IF xEmergenciaOK THEN
	//se nao tiver bloqueado
	IF NOT xBloqueado THEN
		//tudo que da pra considerar uma falha
		IF (NOT xFalha) THEN
			IF xLigaManu OR (xLigaManu3S AND NOT Ton3Segundos.q) THEN
				xCmdFWD := TRUE;
			ELSE
				xCmdFWD := FALSE;
			END_IF
		END_IF
	END_IF
END_IF

IF (xReset OR xResetBlocoComunicacao) AND xFalha THEN
	xCmdFWD := xCmdRev := FALSE;
END_IF

// joga a velo normal nele 
iVelocidade := real_to_int(rSetPoinManu);

//protege contra numeros negativos ou divisao por 0
IF stMotor.Config.xVeloEmPorcentagem THEN
	rSetPoinManu := 100;

	IF stMotor.Config.rVeloEmPorcentagem_VeloMax < 0.1 THEN
		stMotor.Config.rVeloEmPorcentagem_VeloMax := 1;
	END_IF

	iVelocidade := TO_INT((rSetPoinManu * stMotor.Config.rVeloEmPorcentagem_VeloMax) / 100);
END_IF

IF stMotor.Config.xVeloEmMetroPMin THEN
	//rSetPoinManu := 1800;
	//protege contra numeros negativos ou divisao por 0
	IF stMotor.Config.rVeloEmMetroPMin_Conversao < 0.1 THEN
		stMotor.Config.rVeloEmMetroPMin_Conversao := 1;
	END_IF

	iVelocidade := 1800;//TO_INT((rSetPoinManu * 1800) / stMotor.Config.rVeloEmMetroPMin_Conversao);
END_IF

// se tiver que inverte a velo e tiver comissionado
IF stMotor.Config.xInverteSentido THEN
	//se o operador meter uma velo negativva nao da BO
	IF iVelocidade < 0 THEN
		iVelocidade := iVelocidade;
	ELSE
		iVelocidade := iVelocidade * -1;
	END_IF

END_IF

xLigado := (xCmdFwd OR xCmdRev) AND xFazendoComissionamento;
END_ACTION

ACTION Falhas:

xResetParaInversor := xReset OR xResetBlocoComunicacao;

IF xReset OR xResetBlocoComunicacao THEN
	xFalhaContatora := FALSE;
	xFalhaPartidaSoft := FALSE;
END_IF

rtVoltouOnline(CLK := xInversorOnline, Q =>);

IF rtVoltouOnline.q THEN
	xFalha	:= FALSE;
	xReset	:= TRUE;
END_IF

TON_Partida(IN := ((xCmdFwd OR xCmdRev) AND NOT ((xContatorLigado OR xByPassContator)) AND xTemContatora),
			PT := REAL_TO_TIME(stMotor.Config.rTempoFeedBackContator * 1000),
			Q =>,
			ET =>);

IF TON_Partida.q THEN
	xFalhaContatora := TRUE;
END_IF

// as condiçoes que geram falha
xFalha := FALSE;

// se nao vier o sinal da contatora
IF xFalhaContatora THEN
	xFalha := TRUE OR xFalha;
END_IF

//Disjuntor desarmado
IF (NOT xDisjuntorOK AND NOT xByPassDisjuntor) AND xTemDisjuntor THEN
	xFalha := TRUE OR xFalha;
END_IF

// se o inversor nao ficar online
IF ((xTemInversor OR xTemTeSysU) AND (NOT xInversorOnline AND NOT xBypassRede)) THEN
	xFalha := TRUE OR xFalha;
END_IF

//se o inversor entrar em falha
IF ((xTemInversor OR xTemTeSysU) AND (xFalhaInversor AND NOT xBypassRede)) THEN
	xFalha := TRUE OR xFalha;
END_IF

//se o inversor entrar em falha
IF (xTemContatoInversorOK AND ((NOT xContatoInversorOK) AND NOT xBypassContatoInversorOK)) THEN
	xFalha := TRUE OR xFalha;
END_IF

//se o freio nao vier
IF (NOT xFreioOK AND NOT xBypassFreio) AND stMotor.Config.xTemFreio THEN
	xFalha := TRUE OR xFalha;
END_IF


TON_soft
	(
		IN := (xCmdFwd OR xCmdRev) AND NOT (xContatoRodandoSoft OR xBypassContatorunSoft) AND stMotor.Config.xTemSoft,
			PT := REAL_TO_TIME(stMotor.Config.rTempoDeRampaSoft * 1000),
			Q =>,
			ET =>);

IF TON_soft.q THEN
	xFalhaPartidaSoft := TRUE;
END_IF

IF xFalhaPartidaSoft THEN
	xFalha := TRUE OR xFalha;
END_IF

IF xSoftEmFalhaCOM AND NOT xBypassSoftEmFalhaCOM THEN
	xFalha := TRUE OR xFalha;
END_IF

//se o inversor entrar em falha
IF ((xContatoFalhaSoft) AND NOT stMotor.Config.xBypassContatoFalhaSoft) AND stMotor.Config.xTemSoft THEN
	xFalha := TRUE OR xFalha;
END_IF

//se foi detectada uma falta de fase
IF NOT xFaltaDeFaseOk THEN
	xFalha := TRUE OR xFalha;
END_IF
END_ACTION

METHOD FB_init : BOOL
VAR_INPUT
	bInitRetains	: BOOL;	// if TRUE, the retain variables are initialized (warm start / cold start)
	bInCopyCode		: BOOL;	// if TRUE, the instance afterwards gets moved into the copy code (online change)
END_VAR

(*
IF bInCopyCode THEN
	
	IF CHK_REAL(stMotor.Config.iSetPoinManu) <> 0 THEN
		stMotor.Config.iSetPoinManu := 0;
	END_IF
	
	IF CHK_REAL(stMotor.Config.rCorrente_Comissionada) <> 0 THEN
		stMotor.Config.rCorrente_Comissionada := 0;
	END_IF
	
	IF CHK_REAL(stMotor.Config.rSetPoinAuto) <> 0 THEN
		stMotor.Config.rSetPoinAuto := 0;
	END_IF
	
	IF CHK_REAL(stMotor.Config.rTempoFeedBackContator) <> 0 THEN
		stMotor.Config.rTempoFeedBackContator := 0;
	END_IF
	
	IF CHK_REAL(stMotor.Config.rTempoProxMotor) <> 0 THEN
		stMotor.Config.rTempoProxMotor := 0;
	END_IF
	
	IF CHK_REAL(stMotor.Config.rTempoTrocaSentidoDeMarcha) <> 0 THEN
		stMotor.Config.rTempoTrocaSentidoDeMarcha := 0;
	END_IF
	
	IF CHK_REAL(stMotor.Config.rVeloEmMetroPMin_Conversao) <> 0 THEN
		stMotor.Config.rVeloEmMetroPMin_Conversao := 0;
	END_IF
	
	IF (stMotor.Config.xByPassContator) <> TRUE AND (stMotor.Config.xByPassContator) <> FALSE THEN
		stMotor.Config.xByPassContator := FALSE;
	END_IF
	
	IF (stMotor.Config.xByPassDisjuntor) <> TRUE AND (stMotor.Config.xByPassDisjuntor) <> FALSE THEN
		stMotor.Config.xByPassDisjuntor := FALSE;
	END_IF
	
	IF (stMotor.Config.xBypassRede) <> TRUE AND (stMotor.Config.xBypassRede) <> FALSE THEN
		stMotor.Config.xBypassRede := FALSE;
	END_IF
	
	IF (stMotor.Config.xComissionado_Corrente) <> TRUE AND (stMotor.Config.xComissionado_Corrente) <> FALSE THEN
		stMotor.Config.xComissionado_Corrente := FALSE;
	END_IF
	
	IF (stMotor.Config.xComissionado_Sentido) <> TRUE AND (stMotor.Config.xComissionado_Sentido) <> FALSE THEN
		stMotor.Config.xComissionado_Sentido := FALSE;
	END_IF
	
	IF (stMotor.Config.xComissionado_Velo) <> TRUE AND (stMotor.Config.xComissionado_Velo) <> FALSE THEN
		stMotor.Config.xComissionado_Velo := FALSE;
	END_IF
	
	IF (stMotor.Config.xInverteSentido) <> TRUE AND (stMotor.Config.xInverteSentido) <> FALSE THEN
		stMotor.Config.xInverteSentido := FALSE;
	END_IF
	
	IF (stMotor.Config.xTemReversao) <> TRUE AND (stMotor.Config.xTemReversao) <> FALSE THEN
		stMotor.Config.xTemReversao := FALSE;
	END_IF
	
	IF (stMotor.Config.xVeloEmMetroPMin) <> TRUE AND (stMotor.Config.xVeloEmMetroPMin) <> FALSE THEN
		stMotor.Config.xVeloEmMetroPMin := FALSE;
	END_IF
	
	IF (stMotor.Config.xVeloEmPorcentagem) <> TRUE AND (stMotor.Config.xVeloEmPorcentagem) <> FALSE THEN
		stMotor.Config.xVeloEmPorcentagem := FALSE;
	END_IF

END_IF
*)
END_METHOD

ACTION FirstScan:




//Ultima_stMotor		:= stMotor;
rSetPoinManu		:= stMotor.Config.rSetPoinManu;
rSetPoinAuto		:= stMotor.Config.rSetPoinAuto;
xByPassContator		:= stMotor.Config.xByPassContator;
xByPassDisjuntor	:= stMotor.Config.xByPassDisjuntor;

FOR i := 0 TO 23 DO
	stMotor.KPI[i].stGraficoIHM[0].x := 'Desligado';
	stMotor.KPI[i].stGraficoIHM[0].sCor := '#555555';
	stMotor.KPI[i].stGraficoIHM[0].y := 100;
	
	stMotor.KPI[i].stGraficoIHM[1].x := 'Ligado';
	stMotor.KPI[i].stGraficoIHM[1].sCor := '#F1F1F1';
	
	stMotor.KPI[i].stGraficoIHM[2].x := 'Interlok';
	stMotor.KPI[i].stGraficoIHM[2].sCor := '#FFFF00';
	
	stMotor.KPI[i].stGraficoIHM[3].x := 'Falha';
	stMotor.KPI[i].stGraficoIHM[3].sCor := '#FF0000';
	
	stMotor.KPI[i].stGraficoIHM[4].x := 'Emergencia';
	stMotor.KPI[i].stGraficoIHM[4].sCor := '#CC0000';
END_FOR
END_ACTION

ACTION Horimetro:
(*// aqui ta o lendario codigo que no incendo do frigorifico de rolandia diminuiu de 30 para 15 o uso da CPU, chupa mundo
// muito inificiente //Total chad de codigo
systime(timeLoDw => currentTime.dwLowDateTime, timeHiDW => currentTime.dwHighDateTime);

dtAux := FILETIME_TO_DT(currentTime)-(T#3H);
timeStructAux := DT_TO_SYSTEMTIME(dtAux);
*)

fbHorimetro(xConta := stMotor.Sa.xCmdFwd OR stMotor.Sa.xCmdRev,
			xReset := stHoraAgora.wDay <> wDiaAnterior,
			Tempo => tHorimetro,
			stHoraAgora := stHoraAgora);

wDiaAnterior := stHoraAgora.wDay;

sHorimetro := F_TempoEmStringAteHoras
	(
		Tempo := tHorimetro,
			xMostraHoras := TRUE,
			xMostraMinutos := TRUE,
			xMostraSegundos := TRUE,
			xMostraMilisegundos := FALSE,
			xCascata := FALSE);

stMotor.Sa.sHorimetro	:= sHorimetro;
stMotor.Sa.tHorimetro	:= tHorimetro;
END_ACTION

ACTION KPI:

rtLigou(CLK:=xLigado);
IF rtLigou.q THEN
	IF xLigado THEN
		stMotor.KPI[0].iVezesLigado := stMotor.KPI[0].iVezesLigado + 1;
	ELSE
		stMotor.KPI[0].iVezesdesligado := stMotor.KPI[0].iVezesdesligado + 1;
	END_IF
END_IF

rtfalha(CLK:=xFalha);
IF rtfalha.q THEN
	stMotor.KPI[0].iVezesFalha := stMotor.KPI[0].iVezesFalha + 1;
END_IF

rtEmergencia(CLK:=xEmergenciaOK);
IF rtEmergencia.q THEN
	stMotor.KPI[0].iVezesEmergencia := stMotor.KPI[0].iVezesEmergencia + 1;
END_IF

rtInterlock(CLK:=xParadoPorInterlock);
IF rtInterlock.q THEN
	stMotor.KPI[0].iVezesInterlock := stMotor.KPI[0].iVezesInterlock + 1;
END_IF



IF wSegAnterior <> stHoraAgora.wSecond THEN

	IF xFalha AND xEmergenciaOK THEN
		stMotor.KPI[0].rPorcFalha	:= stMotor.KPI[0].rPorcFalha + 0.027777;
		stMotor.KPI[0].tFalha		:= stMotor.KPI[0].tFalha + T#1S;
	END_IF

	IF NOT xEmergenciaOK THEN
		stMotor.KPI[0].rPorcEmergencia	:= stMotor.KPI[0].rPorcEmergencia + 0.027777;
		stMotor.KPI[0].tEmergencia		:= stMotor.KPI[0].tEmergencia + T#1S;
	END_IF

	IF xParadoPorInterlock THEN
		stMotor.KPI[0].rPorcInterlock	:= stMotor.KPI[0].rPorcInterlock + 0.027777;
		stMotor.KPI[0].tInterlock		:= stMotor.KPI[0].tInterlock + T#1S;
	END_IF

	IF xCmdFwd THEN
		stMotor.KPI[0].rPorcLigado	:= stMotor.KPI[0].rPorcLigado + 0.027777;
		stMotor.KPI[0].tLigado		:= stMotor.KPI[0].tLigado + T#1S;
	END_IF
	
	
	// Pro OEE Fechar ele precisa considerar so o tempo que ele deveria estar ligado
	IF xLigaAuto THEN // Para o OEE
		tTempoComxLigaAuto		:= tTempoComxLigaAuto + T#1S;
	END_IF
	
	IF xLigaAuto AND NOT xEmergenciaOK THEN // Para o OEE
		tXligaEEmergencia		:= tXligaEEmergencia + T#1S;
	END_IF
	
	IF xLigaAuto AND xParadoPorInterlock THEN // Para o OEE
		tXligaEInterlock		:= tXligaEInterlock + T#1S;
	END_IF
	
	IF xLigaAuto AND xFalha AND xEmergenciaOK THEN // Para o OEE
		tXligaEFalha			:= tXligaEFalha + T#1S;
	END_IF
	
	

	stMotor.KPI[0].rPorcDesligado :=
		100 - stMotor.KPI[0].rPorcLigado - stMotor.KPI[0].rPorcInterlock - stMotor.KPI[0].rPorcEmergencia - stMotor.KPI[0].rPorcFalha;

	stMotor.KPI[0].tDesligado :=
		T#1H - stMotor.KPI[0].tLigado - stMotor.KPI[0].tInterlock - stMotor.KPI[0].tEmergencia - stMotor.KPI[0].tFalha;
		
	rAux := DINT_TO_REAL(TRUNC(stMotor.KPI[0].rPorcDesligado*100));
	stMotor.KPI[0].stGraficoIHM[0].y := rAux/100;
	rAux := DINT_TO_REAL(TRUNC(stMotor.KPI[0].rPorcLigado*100));
	stMotor.KPI[0].stGraficoIHM[1].y := rAux/100;
	rAux := DINT_TO_REAL(TRUNC(stMotor.KPI[0].rPorcInterlock*100));
	stMotor.KPI[0].stGraficoIHM[2].y := rAux/100;
	rAux := DINT_TO_REAL(TRUNC(stMotor.KPI[0].rPorcFalha*100));
	stMotor.KPI[0].stGraficoIHM[3].y := rAux/100;
	rAux := DINT_TO_REAL(TRUNC(stMotor.KPI[0].rPorcEmergencia*100));
	stMotor.KPI[0].stGraficoIHM[4].y := rAux/100;
	


END_IF

IF whoraAnterior <> stHoraAgora.wHour THEN
	
	//OEE
	udiLigado 		:= TIME_TO_UDINT(tTempoComxLigaAuto);
	udiFalha 		:= TIME_TO_UDINT(tXligaEFalha);
	udiEmergencia 	:= TIME_TO_UDINT(tXligaEEmergencia);
	udiinterlock 	:= TIME_TO_UDINT(tXligaEInterlock);
	
	
	rAux1 := (udiLigado-udiFalha);
	IF udiLigado <> 0 THEN
		rAux1 := rAux1/udiLigado; // disponibilidade em valor
		stMotor.KPI[0].rDisponibilidade := rAux1 * 100;
	ELSE
		stMotor.KPI[0].rDisponibilidade := 0;
	END_IF
	
	rAux1 := (udiLigado-udiFalha-udiEmergencia-udiinterlock);
	rAux2 := (udiLigado-udiFalha);
	IF rAux2 <> 0 THEN
		rAux1 := rAux1/rAux2; // Performace em valor
		stMotor.KPI[0].rPerformace := rAux1 * 100;
	ELSE
		stMotor.KPI[0].rPerformace := 0;
	END_IF
	
	
	stMotor.KPI[0].rQualidade := 100;
	stMotor.KPI[0].rOEE := (stMotor.KPI[0].rDisponibilidade * stMotor.KPI[0].rPerformace * stMotor.KPI[0].rQualidade) / 10000;
	
	
	
	stMotor.KPI[0].stGraficoDisponibilidade[0].x := 'Disponivel';
	stMotor.KPI[0].stGraficoDisponibilidade[0].sCor := '#32CD32';
	stMotor.KPI[0].stGraficoDisponibilidade[0].label := ' ';
	stMotor.KPI[0].stGraficoDisponibilidade[0].y := stMotor.KPI[0].rDisponibilidade;
	
	stMotor.KPI[0].stGraficoDisponibilidade[0].x := 'Indisponivel';
	stMotor.KPI[0].stGraficoDisponibilidade[0].sCor := '#FFFFFF00';
	stMotor.KPI[0].stGraficoDisponibilidade[0].label := ' ';
	stMotor.KPI[0].stGraficoDisponibilidade[0].y := 100 - stMotor.KPI[0].rDisponibilidade;
	
	
	stMotor.KPI[0].stGraficoPerformace[0].x := 'Performando';
	stMotor.KPI[0].stGraficoPerformace[0].sCor := '#32CD32';
	stMotor.KPI[0].stGraficoPerformace[0].label := ' ';
	stMotor.KPI[0].stGraficoPerformace[0].y := stMotor.KPI[0].rPerformace;
	
	stMotor.KPI[0].stGraficoPerformace[0].x := 'Não performando';
	stMotor.KPI[0].stGraficoPerformace[0].sCor := '#FFFFFF00';
	stMotor.KPI[0].stGraficoPerformace[0].label := ' ';
	stMotor.KPI[0].stGraficoPerformace[0].y := 100 - stMotor.KPI[0].rPerformace;
	
	
	stMotor.KPI[0].stGraficoQualidade[0].x := 'Qualidade';
	stMotor.KPI[0].stGraficoQualidade[0].sCor := '#32CD32';
	stMotor.KPI[0].stGraficoQualidade[0].label := ' ';
	stMotor.KPI[0].stGraficoQualidade[0].y := stMotor.KPI[0].rQualidade;
	
	stMotor.KPI[0].stGraficoQualidade[0].x := 'Mal qualidade';
	stMotor.KPI[0].stGraficoQualidade[0].sCor := '#FFFFFF00';
	stMotor.KPI[0].stGraficoQualidade[0].label := ' ';
	stMotor.KPI[0].stGraficoQualidade[0].y := 100 - stMotor.KPI[0].rQualidade;
	
	
	stMotor.KPI[0].stGraficoOEE[0].x := 'OEE';
	stMotor.KPI[0].stGraficoOEE[0].sCor := '#32CD32';
	stMotor.KPI[0].stGraficoOEE[0].label := ' ';
	stMotor.KPI[0].stGraficoOEE[0].y := stMotor.KPI[0].rOEE;
	
	stMotor.KPI[0].stGraficoOEE[0].x := 'OEE ruim';
	stMotor.KPI[0].stGraficoOEE[0].sCor := '#FFFFFF00';
	stMotor.KPI[0].stGraficoOEE[0].label := ' ';
	stMotor.KPI[0].stGraficoOEE[0].y := 100 - stMotor.KPI[0].rOEE;
	
	
	
	
	//KPI NORMAL


	FOR i := 23 TO 1 BY -1 DO
		stMotor.KPI[i] := stMotor.KPI[i - 1];
	END_FOR

	stMotor.KPI[0] := kpiVazio;
	tTempoComxLigaAuto := T#0S;
	tXligaEEmergencia := T#0S;
	tXligaEFalha := T#0S;
	tXligaEInterlock := T#0S;
	
	stMotor.KPI[0].stGraficoIHM[0].x := 'Desligado';
	stMotor.KPI[0].stGraficoIHM[0].sCor := '#555555';
	stMotor.KPI[0].stGraficoIHM[0].label := ' ';
	stMotor.KPI[0].stGraficoIHM[0].y := 100;
	
	stMotor.KPI[0].stGraficoIHM[1].x := 'Ligado';
	stMotor.KPI[0].stGraficoIHM[1].label := ' ';
	stMotor.KPI[0].stGraficoIHM[1].sCor := '#F1F1F1';
	
	stMotor.KPI[0].stGraficoIHM[2].x := 'Interlok';
	stMotor.KPI[0].stGraficoIHM[2].label := ' ';
	stMotor.KPI[0].stGraficoIHM[2].sCor := '#FFFF00';
	
	stMotor.KPI[0].stGraficoIHM[3].x := 'Falha';
	stMotor.KPI[0].stGraficoIHM[3].label := ' ';
	stMotor.KPI[0].stGraficoIHM[3].sCor := '#FF0000';
	
	stMotor.KPI[0].stGraficoIHM[4].x := 'Emergencia';
	stMotor.KPI[0].stGraficoIHM[4].label := ' ';
	stMotor.KPI[0].stGraficoIHM[4].sCor := '#CC0000';
END_IF

whoraAnterior	:= stHoraAgora.wHour;
wSegAnterior	:= stHoraAgora.wSecond;
END_ACTION

ACTION ProxMotor:

/// Liga prox motor na sequencia

// se tiver o comando pra ligar ele ja manda essa e se tiver inversor ele ajeita ali em baixo
tonLigaProxMotor.IN := (xCmdFwd OR xCmdRev) AND NOT xFalha;

//se tiver inversor
IF xTemInversor AND (xCmdFwd OR xCmdRev) THEN
	//se o inversor mandar que velo ele ta
	IF stMotor.LeiturasInversorIHM.sVelocidadeRPM <> ''
			AND stMotor.LeiturasInversorIHM.sVelocidadeRPM <> 'NA'
			AND stMotor.LeiturasInversorIHM.sVelocidadeRPM <> 'ND' THEN
		tonLigaProxMotor.IN :=xCmdFwd; // AND NOT xFalha;		
	END_IF
END_IF

tonLigaProxMotor(PT := REAL_TO_TIME(stMotor.Config.rTempoProxMotor * 1000), Q => , ET =>);

xNaoLigaProxMotor := NOT tonLigaProxMotor.q;
END_ACTION

ACTION SegurancaReversao:

//Prende eles em falso para o motor esperar trocar o sentido de giro

xTrocandoSentido := FALSE;
//lembrando que tp funciona na base do pulso , entao faz sentido ser assim
tpTrocaSentidoDeRotacao(IN :=, PT := REAL_TO_TIME(stMotor.Config.rTempoTrocaSentidoDeMarcha * 1000), Q =>, ET =>);

IF tpTrocaSentidoDeRotacao.q AND xLigado THEN
	xCmdFWD := xCmdRev	:= FALSE;
	xTrocandoSentido	:= TRUE;
END_IF

//Controle caso ele troque o sentido 
tpTrocaSentidoDeRotacao.IN := FALSE;

btTrocouSentidoRotAuto(CLK := xReversoAuto AND stMotor.Config.xTemReversao, Q =>);

IF btTrocouSentidoRotAuto.q THEN
	IF xCmdFwd OR xCmdRev THEN
		IF xAutomaticoManual THEN
			tpTrocaSentidoDeRotacao.IN := TRUE;
		END_IF
	END_IF
END_IF

btTrocouSentidoRotManu(CLK := xReversoManu AND stMotor.Config.xTemReversao, Q =>);

IF btTrocouSentidoRotManu.q THEN
	IF xCmdFwd OR xCmdRev THEN
		IF NOT xAutomaticoManual THEN
			tpTrocaSentidoDeRotacao.IN := TRUE;
		END_IF
	END_IF
END_IF

btTrocouManualAutomatico(CLK := xAutomaticoManual AND stMotor.Config.xTemReversao, Q =>);

IF btTrocouManualAutomatico.q THEN
	IF xReversoAuto <> xReversoManu THEN
		tpTrocaSentidoDeRotacao.IN := TRUE;
	END_IF
END_IF
END_ACTION

ACTION Status:

//STAUTS
IF (NOT xCmdFwd OR NOT xCmdrev) AND NOT xBloqueado AND xEmergenciaOK THEN
	IF xAutomaticoManual THEN
		iStsMotor := 1; // parado em automatico
		sStatus := 'Parado em automatico';
	ELSE
		iStsMotor := 2; // parado em manual
		sStatus := 'Parado em manual';
	END_IF
END_IF

IF (xCmdFwd OR xCmdrev) AND (NOT xBloqueado OR xEmergenciaOK) THEN
	IF xAutomaticoManual THEN
		iStsMotor := 3; // rodando em automatico
		sStatus := 'Rodando em automatico';
	ELSE
		iStsMotor := 4; // rodando em manual
		sStatus := 'Rodando em manual';
	END_IF
END_IF

IF stMotor.En.xLigaHigienizacao AND xHabilitaHigienizacao THEN
	iStsMotor := 18; // Higienização Ligada
	sStatus := 'Rodando Higienização';
END_IF

IF stMotor.En.xLigaHigienizacao AND NOT xHabilitaHigienizacao THEN
	iStsMotor := 17; // Higienização Parado
	sStatus := 'Parado Higienização';
END_IF

IF xParadoPorInterlock THEN
	iStsMotor := 10; // Parado por interlock
	sStatus := 'Parado por interlock';
END_IF

IF xTrocandoSentido THEN
	iStsMotor := 11; // Trocando sentido
	sStatus := 'trocando sentido de giro';
END_IF

IF xBloqueado THEN
	iStsMotor := 5; // bloquado
	sStatus := 'Bloqueado';
END_IF

IF xFalhaContatora THEN
	iStsMotor := 6; // em falha na partida
	sStatus := 'Falha contatora';
END_IF

IF ((xTemInversor OR xTemTeSysU) AND (NOT xInversorOnline AND NOT xBypassRede)) THEN
	iStsMotor := 7; // em inversor offline
	IF xTemInversor THEN
		sStatus := 'Inversor offline';
	ELSE
		sStatus := 'TeSysU offline';
	END_IF
END_IF

IF ((xTemInversor OR xTemTeSysU) AND (xFalhaInversor AND NOT xBypassRede)) THEN
	iStsMotor := 12; // Inversor em falha
	IF xTemInversor THEN
		sStatus := 'Falha COM. inversor';
	ELSE
		sStatus := 'Falha COM. TeSysU';
	END_IF
END_IF

IF (xTemContatoInversorOK AND (NOT (xContatoInversorOK) AND NOT xBypassContatoInversorOK)) THEN
	iStsMotor := 14; // Inversor Sem o contato de OK
	sStatus := 'Falha contato inversor';
END_IF

IF NOT xDisjuntorOK AND NOT xByPassDisjuntor AND xTemDisjuntor THEN
	iStsMotor := 8; // disjuntor desarmado
	sStatus := 'Disjuntor desarmado';
END_IF

IF (stMotor.Config.xTemFreio AND (NOT xFreioOK AND NOT xBypassFreio)) THEN
	iStsMotor := 13; // disjuntor desarmado
	sStatus := 'Disjuntor desarmado';
END_IF

IF xFalhaPartidaSoft THEN
	iStsMotor := 15; // em falha na partida da soft
	sStatus := 'Falha na partida da soft';
END_IF

IF ((xContatoFalhaSoft)) AND stMotor.Config.xTemSoft THEN
	iStsMotor := 16; // em falha na soft
	sStatus := 'Falha contato soft';
END_IF

IF ((xSoftEmFalhaCOM)) AND stMotor.Config.xBypassSoftEmFalhaCOM THEN
	iStsMotor := 19; // em falha na soft
	sStatus := 'Falha COM. soft';
END_IF


IF NOT xFaltaDeFaseOk THEN
	iStsMotor := 20; // Falta de fase detectada
	sStatus := 'falta de fase';
END_IF

IF NOT xEmergenciaOK THEN
	iStsMotor := 9; // emergencia
	sStatus := 'Emergencia';
END_IF
END_ACTION

END_FUNCTION_BLOCK

// POUs/Siemens/SinaSpeed/Sina_SpeedV2
FUNCTION_BLOCK Sina_SpeedV2
VAR_IN_OUT
	motor : st_Partida;
END_VAR
VAR_INPUT
	EnableAxis	:	BOOL;//	0	Non-RETAIN	TRUE	TRUE	TRUE	FALSE	0-->1; 1 = Enable the drive (OFF2 / OFF 3 are 1 in default status) (OFF1 = 0-->1)
	AckError	:	BOOL;//	0	Non-RETAIN	TRUE	TRUE	TRUE	FALSE	1 = Acknowledge drive error
	SpeedSp		:	REAL;//	0.0	Non-retain	True	True	True	False	Speed standardises with the standardisation factor
	RefSpeed	:	REAL;//	0.0	Non-retain	True	True	True	False	Standardisation factor of speed
	ConfigAxis	:	Word_Bits;//	Non-RETAIN	TRUE	TRUE	TRUE	FALSE	binary programmed input TO control all functions in the telegram without its own FUNCTION block input
	HWIDZSW AT %I* 	:	InversorSinaSpeed;//	Non-retain	True	True	True	False	Hardware Identifer set point slot
END_VAR
VAR_OUTPUT
	AxisEnabled	:	BOOL;//	0	Non-RETAIN	TRUE	TRUE	TRUE	FALSE	1 = Drive is enabled
	Lockout		:	BOOL;//	0	Non-RETAIN	TRUE	TRUE	TRUE	FALSE	1 = Drive lockout active
	ActVelocity	:	REAL;//	0.0	Non-RETAIN	TRUE	TRUE	TRUE	FALSE	Actual in [U/MIN]
	Error		:	BOOL;//	0	Non-RETAIN	TRUE	TRUE	TRUE	FALSE	1 = Error  (FB AND Infeed)
	Status		:	WORD;//	0	Non-RETAIN	TRUE	TRUE	TRUE	FALSE	Status output (7002 = FB in operation; 8xxx = error description  - read the manual)
	DiagId		:	WORD;//	16#0000	Non-RETAIN	TRUE	TRUE	TRUE	FALSE	Error codes OF the cyclic system funtion blocks DPWR / DPRD_DAT
	HWIDSTW AT %Q*	:	Inversor_2Words_SinaSpeed;//	Non-retain	True	True	True	False	Hardware Identifer actual value slot
	Corrente 	: REAL;
	Potencia 	: REAL;
	Torque 		: REAL;
	ErroAtual 	: UINT;
END_VAR
VAR
	sxSendBuf	:	sxSendBuf;//		Non-RETAIN	TRUE	TRUE	TRUE	FALSE	Send buffer
	sxRecvBuf	:	sxRecvBuf;//		Non-RETAIN	TRUE	TRUE	TRUE	FALSE	Receive buffer

	piRetSFC	:	INT;//						Status FOR fault analysis
	piCount		:	INT;//							Freely available counter variable 3
	prVelocity	:	REAL;//							velocity
	pdRecvBuf	:	DWORD;//							Buffer OF Recv-Value
	pdSendBuf	:	DWORD;//							Buffer OF Send-Value
	phLAddr		:	InversorSinaSpeed;//							Start addr FROM the I/O process image area OF MOD (DEC) FOR DPWR_DAT/DPRD_DAT
	swSendBuf	:	ARRAY[0..1] OF WORD;//							Sendepuffer
	swRecvBuf	:	ARRAY[0..1] OF WORD;//							Empfangspuffer         Static variables
	
	//Adicionado por Tiago
	xPrimeiroScan : BOOL := TRUE;
END_VAR


//=============================================================================
//SIEMENS AG
//(c)Copyright 2017 All Rights Reserved
//-----------------------------------------------------------------------------
// Library: DriveLib
// Tested with: S7-1516-3 PN/DP V1.8
// Engineering: TIA Portal V14
// Restrictions: -
// Requirements: S7-1200 / S7-1500
// Functionality: cyclic communication between a SINAMICS a PLC.
//                If in HWConfig Std.TLG 1 is projected 2 PZD-words are exchanged
//                in every bus cycle.
//                The parametrisation of these words is described in the manual of the
//                SINAMICS
//=============================================================================

//Adicionado por Tiago
IF xPrimeiroScan THEN
	ConfigAxis.wor := 63;
	xPrimeiroScan := FALSE;
END_IF


EnableAxis := motor.Sa.xCmdFwd;
AckError := motor.Sa.xResetParaInversor;
SpeedSp := motor.Sa.iVelocidade;





Corrente := HWIDZSW.StatusWord2.ui16b * 25.0 / 16384; // 2.5 = parametro interno
Torque := HWIDZSW.StatusWord3.ui16b * 58.36 / 16384; // parametro interno
Potencia := HWIDZSW.StatusWord4.ui16b * 11.0 / 16384; // parametro interno
ErroAtual := HWIDZSW.StatusWord5.ui16b;

motor.LeiturasInversorIHM.sVelocidadeRPM := concat(TO_STRING(F_RetiraCasa(Entrada:= ActVelocity, casa:= 1)),' RPM');
motor.LeiturasInversorIHM.sCorrente := concat(TO_STRING(F_RetiraCasa(Entrada:= Corrente, casa:= 2)),' A');
motor.LeiturasInversorIHM.sTorque := concat(TO_STRING(F_RetiraCasa(Entrada:= Torque, casa:= 2)),' Nm');
motor.LeiturasInversorIHM.sVelocidadeHz := concat(TO_STRING(F_RetiraCasa(Entrada:= Potencia, casa:= 2)),' KW');
motor.LeiturasInversorIHM.sUltimoErro := TO_STRING(DiagId);

// Fim adicionado por tiago

















// Schreibdaten zusammenstellen
// Steuerword aufbereiten

sxSendBuf.STW1.x16b.bBit0 := EnableAxis;
sxSendBuf.STW1.x16b.bBit1 := ConfigAxis.bits.bBit0;
sxSendBuf.STW1.x16b.bBit2 := ConfigAxis.bits.bBit1;
sxSendBuf.STW1.x16b.bBit3 := ConfigAxis.bits.bBit2;
sxSendBuf.STW1.x16b.bBit4 := ConfigAxis.bits.bBit3;
sxSendBuf.STW1.x16b.bBit5 := ConfigAxis.bits.bBit4;
sxSendBuf.STW1.x16b.bBit6 := ConfigAxis.bits.bBit5;
sxSendBuf.STW1.x16b.bBit10 := TRUE;
sxSendBuf.STW1.x16b.bBit11 := ConfigAxis.bits.bBit6;
sxSendBuf.STW1.x16b.bBit7 := AckError;

// Geschwindigkeit
IF RefSpeed <> 0 THEN
  prVelocity := SpeedSp * (16384.0 / RefSpeed);
  // Limit REAL - Variable to INT - Limits
  IF prVelocity > 32767 THEN
    prVelocity := 32767;
  ELSIF prVelocity < -32768 THEN
    prVelocity := -32768;
  ELSE
    ; // not needed
  END_IF;
  sxSendBuf.Velocity.Valor := INT_TO_WORD(REAL_TO_INT(prVelocity));
  
ELSE
  sxSendBuf.Velocity.Valor := 16#0;
END_IF;
swSendBuf[0] := sxSendBuf.STW1.ui16b;
swSendBuf[1] := UDINT_TO_WORD(sxSendBuf.Velocity.Valor);

//Prozessdaten zur Signalbaugruppe schreiben
(*
piRetSFC := DPWR_DAT(LADDR := HWIDSTW,
                      RECORD := swSendBuf);
*)

piRetSFC := 0;

HWIDSTW.StatusWord0.ui16b := swSendBuf[0];
HWIDSTW.StatusWord1.ui16b := swSendBuf[1];





// Fehler der RÃ¼ckmeldung ausgeben
DiagId := INT_TO_WORD(piRetSFC);

//kein Fehler beim Schreiben
IF piRetSFC = 0 THEN
  
  //kein Fehler beim Schreiben
  IF piRetSFC = 0 THEN
    
    //Prozessdaten von der Signalbaugruppe lesen
	(*
    #piRetSFC := DPRD_DAT(LADDR := #HWIDZSW,
                          RECORD => #swRecvBuf);
						  *)
	
	piRetSFC := 0;
						  
	swRecvBuf[0] := HWIDZSW.StatusWord0.ui16b;
	swRecvBuf[1] := HWIDZSW.StatusWord1.ui16b;			
    
    // Fehler der RÃ¼ckmeldung ausgeben
    DiagId := INT_TO_WORD(piRetSFC);
  END_IF;
  
  //Fehler beim Lesen (Profibus-Kommunikation unterbrochen)
  IF piRetSFC <> 0 THEN
    
    // Fehler
    Error := TRUE;
    Status := 16#8600;
    
    // Zustandsworte lÃ¶schen
    sxRecvBuf.ZSW1.x16b.bBit8 := 0;
    sxRecvBuf.ZSW1.x16b.bBit9 := 0;
    sxRecvBuf.ZSW1.x16b.bBit10 := 0;
    sxRecvBuf.ZSW1.x16b.bBit11 := 0;
    sxRecvBuf.ZSW1.x16b.bBit12 := 0;
    sxRecvBuf.ZSW1.x16b.bBit13 := 0;
    sxRecvBuf.ZSW1.x16b.bBit14 := 0;
    sxRecvBuf.ZSW1.x16b.bBit15 := 0;
    sxRecvBuf.ZSW1.x16b.bBit0 := 0;
    sxRecvBuf.ZSW1.x16b.bBit1 := 0;
    sxRecvBuf.ZSW1.x16b.bBit2 := 0;
    sxRecvBuf.ZSW1.x16b.bBit3 := 0;
    sxRecvBuf.ZSW1.x16b.bBit4 := 0;
    sxRecvBuf.ZSW1.x16b.bBit5 := 0;
    sxRecvBuf.ZSW1.x16b.bBit6 := 0;
    sxRecvBuf.ZSW1.x16b.bBit7 := 0;
    
    
    (*#sxRecvBuf.sxZSW1.SpDev   := 0;
    #sxRecvBuf.sxZSW1.Pcd     := 0;
    #sxRecvBuf.sxZSW1.Comp    := 0;
    #sxRecvBuf.sxZSW1.CurLim  := 0;
    #sxRecvBuf.sxZSW1.Brake   := 0;
    #sxRecvBuf.sxZSW1.Motover := 0;
    #sxRecvBuf.sxZSW1.Dir     := 0;
    #sxRecvBuf.sxZSW1.Invover := 0;
    #sxRecvBuf.sxZSW1.Rts     := 0;
    #sxRecvBuf.sxZSW1.Rdy     := 0;
    #sxRecvBuf.sxZSW1.IOp     := 0;
    #sxRecvBuf.sxZSW1.Fault   := 0;
    #sxRecvBuf.sxZSW1.NoOff2  := 0;
    #sxRecvBuf.sxZSW1.NoOff3  := 0;
    #sxRecvBuf.sxZSW1.Inhibit := 0;
    #sxRecvBuf.sxZSW1.Alarm   := 0;*)
    
    sxRecvBuf.Velocity.Valor := 0;
    
    // Werte auslesen
  ELSE
    sxRecvBuf.ZSW1.ui16b := swRecvBuf[0];
    sxRecvBuf.Velocity.Valor := swRecvBuf[1];
    
    // ZSW1 aufbereiten                       
    AxisEnabled := sxRecvBuf.ZSW1.x16b.bBit2;
    Error := sxRecvBuf.ZSW1.x16b.bBit3 OR sxRecvBuf.ZSW1.x16b.bBit6;
    Lockout := sxRecvBuf.ZSW1.x16b.bBit6;
    
    // Fehler auswerten
    IF sxRecvBuf.ZSW1.x16b.bBit3 THEN
      Status := 16#8401;
    ELSIF sxRecvBuf.ZSW1.x16b.bBit6 THEN
      Status := 16#8402;
    ELSE
      Status := 16#7002;
    END_IF;
    
    (*#Busy       := #sxRecvBuf.sxZSW1.IOp;
    #Error      := #sxRecvBuf.sxZSW1.Fault OR #sxRecvBuf.sxZSW1.Inhibit;
    #PwrInhibit := #sxRecvBuf.sxZSW1.Inhibit;            

    // Fehler auswerten
    IF #sxRecvBuf.sxZSW1.Fault THEN
        #ErrorId := 1;
    ELSIF #sxRecvBuf.sxZSW1.Inhibit THEN 
        #ErrorId := 2;
    ELSE
        #ErrorId := 0;    
    END_IF;*)
    
    // Geschwindigkeit
    IF RefSpeed <> 0 THEN
      ActVelocity := UDINT_TO_REAL((sxRecvBuf.Velocity.Valor)) / (16384.0 / RefSpeed);
    ELSE
      ActVelocity := 0.0;
    END_IF;
  END_IF;
ELSE
      
  // Fehler
  Error := TRUE;
  Status := 16#8601;
    
END_IF;

END_FUNCTION_BLOCK

// POUs/Siemens/Sina_posV2
FUNCTION_BLOCK Sina_posV2
VAR_INPUT
	ModePos				: INT;					//Settings of the mode
	EnableAxis			: BOOL;					//	0	Non-RETAIN	TRUE	TRUE	TRUE	FALSE	1 = Enable the drive
	CancelTraversing	: BOOL	:= TRUE;		//	Non-RETAIN	TRUE	TRUE	TRUE	FALSE	0 = Reject active traverse task
	IntermediateStop	: BOOL	:= TRUE;		//	Non-RETAIN	TRUE	TRUE	TRUE	FALSE	0 = Intermediate STOP OF traverse command
	Positive			: BOOL;					//	0	Non-RETAIN	TRUE	TRUE	TRUE	FALSE	1 = Direction positive
	Negative			: BOOL;					//	0	Non-RETAIN	TRUE	TRUE	TRUE	FALSE	1 = Direction negative
	Jog1				: BOOL;					//	0	Non-RETAIN	TRUE	TRUE	TRUE	FALSE	1 = Use jog 1 (direction / speed)
	Jog2				: BOOL;					//	0	Non-RETAIN	TRUE	TRUE	TRUE	FALSE	1 = Use jog 2 (direction / speed)
	FlyRef				: BOOL;					//	0	Non-RETAIN	TRUE	TRUE	TRUE	FALSE	1 = Start flying REFERENCE FUNCTION
	AckError			: BOOL;					//	0	Non-RETAIN	TRUE	TRUE	TRUE	FALSE	1  = Acknowledge OF errors
	ExecuteMode			: BOOL;					//	0	Non-RETAIN	TRUE	TRUE	TRUE	FALSE	0-->1 = Start the mode
	Position			: DINT;					//	0	Non-RETAIN	TRUE	TRUE	TRUE	FALSE	Position OF the MDI mode OR setting OF traversing block
	Velocity			: DINT;					//	0	Non-RETAIN	TRUE	TRUE	TRUE	FALSE	MDI velocity
	OverV				: INT	:= 100;			//	Non-RETAIN	TRUE	TRUE	TRUE	FALSE	Override OF  velocity in [%] --> 4000h=100%
	OverAcc				: INT	:= 100;			//	Non-RETAIN	TRUE	TRUE	TRUE	FALSE	Override OF acceleration in [%] --> 4000h=100%
	OverDec				: INT	:= 100;			//	Non-RETAIN	TRUE	TRUE	TRUE	FALSE	Override OF deceleration in [%] --> 4000h=100%
	ConfigEPos			: u16b;					//	Non-RETAIN	TRUE	TRUE	TRUE	FALSE	binary programmed input TO control all functions in the telegram without its own FUNCTION block input
	ConfigEPos2			: u16b;					//	Non-RETAIN	TRUE	TRUE	TRUE	FALSE	binary programmed input TO control all functions in the telegram without its own FUNCTION block input
	HWIDZSW				: InversorSinaSpeed;	//	0	Non-RETAIN	TRUE	TRUE	TRUE	FALSE	Hardware Identifer actual value slot
END_VAR
VAR_OUTPUT
	AxisEnabled	: BOOL;					//	0	Non-RETAIN	TRUE	TRUE	TRUE	FALSE	1= Axis in operation
	AxisPosOk	: BOOL;					//	0	Non-RETAIN	TRUE	TRUE	TRUE	FALSE	1= Position setpoint reached
	AxisRef		: BOOL;					//	0	Non-RETAIN	TRUE	TRUE	TRUE	FALSE	1= REFERENCE point set
	AxisWarn	: BOOL;					//	0	Non-RETAIN	TRUE	TRUE	TRUE	FALSE	1= Axis alarm / warning present
	AxisError	: BOOL;					//	0	Non-RETAIN	TRUE	TRUE	TRUE	FALSE	1= Axis fault present
	Lockout		: BOOL;					//	0	Non-RETAIN	TRUE	TRUE	TRUE	FALSE	1= Axis in lockout state
	ActVelocity	: DINT;					//	0	Non-RETAIN	TRUE	TRUE	TRUE	FALSE	Actual drive speed (has TO be normed with p2000 --> 40000000h = 100%)
	ActPosition	: DINT;					//	0	Non-RETAIN	TRUE	TRUE	TRUE	FALSE	Actual position in [LU]
	ActMode		: INT;					//	0	Non-RETAIN	TRUE	TRUE	TRUE	FALSE	Active EPos mode
	EPosZSW1	: WORD;					//	0	Non-RETAIN	TRUE	TRUE	TRUE	FALSE	Status OF EPOS ZSW1
	EPosZSW2	: WORD;					//	0	Non-RETAIN	TRUE	TRUE	TRUE	FALSE	Status OF EPOS ZSW2
	ActWarn		: WORD;					//	0	Non-RETAIN	TRUE	TRUE	TRUE	FALSE	Actual number OF warning
	ActFault	: WORD;					//	0	Non-RETAIN	TRUE	TRUE	TRUE	FALSE	Actual number OF error
	Error		: BOOL;					//	0	Non-RETAIN	TRUE	TRUE	TRUE	FALSE	1 = Error  (FB AND Infeed)
	Status		: WORD;					//	0	Non-RETAIN	TRUE	TRUE	TRUE	FALSE	Status output (7002 = FB in operation; 8xxx = error description  - read the manual)
	DiagID		: WORD;					//	0	Non-RETAIN	TRUE	TRUE	TRUE	FALSE	Error codes OF the cyclic system funtion blocks DPWR / DPRD_DAT
	HWIDSTW		: InversorSinaSpeed;	//	0	Non-RETAIN	TRUE	TRUE	TRUE	FALSE	Hardware Identifer set point slot
END_VAR
VAR
	sbOff1Edge		: BOOL;				//	0	Non-RETAIN	TRUE	TRUE	TRUE	FALSE	Positive edge OF starting OR stopping the device
	sbOff1			: BOOL;				//	0	Non-RETAIN	TRUE	TRUE	TRUE	FALSE	Starting OR stopping the device
	sbExecuteEdge	: BOOL;				//	0	Non-RETAIN	TRUE	TRUE	TRUE	FALSE	Positive edge OF activate traversing block
	sbExecute		: BOOL;				//	0	Non-RETAIN	TRUE	TRUE	TRUE	FALSE	Activate traversing block
	sbRefTypEdge	: BOOL;				//	0	Non-RETAIN	TRUE	TRUE	TRUE	FALSE	Positive edge OF referencing TYPE "flying reference"
	sbRefTyp		: BOOL;				//	0	Non-RETAIN	TRUE	TRUE	TRUE	FALSE	Referencing TYPE "flying reference"
	sbMdiStart		: BOOL;				//	0	Non-RETAIN	TRUE	TRUE	TRUE	FALSE	Direct setpoint input / MDI - start
	sbMdiStartEdge	: BOOL;				//	0	Non-RETAIN	TRUE	TRUE	TRUE	FALSE	Positive edge OF direct setpoint input / MDI - start
	sbRefStart		: BOOL;				//	0	Non-RETAIN	TRUE	TRUE	TRUE	FALSE	Referencing start
	sbJogInc		: BOOL;				//	0	Non-RETAIN	TRUE	TRUE	TRUE	FALSE	Jogging incremental
	sbReady			: BOOL;				//	0	Non-RETAIN	TRUE	TRUE	TRUE	FALSE	Ready TO power up / TO start
	sbIOp			: BOOL;				//	0	Non-RETAIN	TRUE	TRUE	TRUE	FALSE	Ready TO operate
	sbAccel			: BOOL;				//	0	Non-RETAIN	TRUE	TRUE	TRUE	FALSE	Axis accelerating
	sbDecel			: BOOL;				//	0	Non-RETAIN	TRUE	TRUE	TRUE	FALSE	Axis decelerating
	sbAlarm			: BOOL;				//	0	Non-RETAIN	TRUE	TRUE	TRUE	FALSE	Alarm / Warnung present
	sbFault			: BOOL;				//	0	Non-RETAIN	TRUE	TRUE	TRUE	FALSE	Fault present
	sbFWD			: BOOL;				//	0	Non-RETAIN	TRUE	TRUE	TRUE	FALSE	Axis drives forwards
	sbBWD			: BOOL;				//	0	Non-RETAIN	TRUE	TRUE	TRUE	FALSE	Axis drives backwards
	sbBusy			: BOOL;				//	0	Non-RETAIN	TRUE	TRUE	TRUE	FALSE	Mode OF operation is explained
	swStatus		: WORD	:= 16#0000;	//	Non-RETAIN	TRUE	TRUE	TRUE	FALSE	Mode OF operation disturbance
	swEPosZSW1		: WORD	:= 16#0000;	//	Non-RETAIN	TRUE	TRUE	TRUE	FALSE	Status OF EPOS ZSW1
	swEPosZSW2		: WORD	:= 16#0000;	//	Non-RETAIN	TRUE	TRUE	TRUE	FALSE	Status OF EPOS ZSW2
	siExecuteCyc	: INT;				//	0	Non-RETAIN	TRUE	TRUE	TRUE	FALSE	Counter OF runcycle OF active traversing block
	siRefTypCyc		: INT;				//	0	Non-RETAIN	TRUE	TRUE	TRUE	FALSE	Counter OF runcycle OF referencing TYPE "flying reference"
	siJogIncCyc		: INT;				//	0	Non-RETAIN	TRUE	TRUE	TRUE	FALSE	Counter OF runcycle OF jogging incremental
	siMdiStartCyc	: INT;				//	0	Non-RETAIN	TRUE	TRUE	TRUE	FALSE	Counter OF runcycle OF direct setpoint input / MDI - start
	siRefActRetry	: INT;				//	0	Non-RETAIN	TRUE	TRUE	TRUE	FALSE	Counter OF retry OF REFERENCE point approach active
	siModePos		: INT;				//	0	Non-RETAIN	TRUE	TRUE	TRUE	FALSE	Setting OF mode
	siModePosMax	: INT	:= 14;		//	Non-RETAIN	TRUE	TRUE	TRUE	FALSE	MAX. count OF mode
	siCycWait		: INT	:= 5;		//	Non-RETAIN	TRUE	TRUE	TRUE	FALSE	Counter OF cycle OF waiting
	siRetryMax		: INT	:= 15;		//	Non-RETAIN	TRUE	TRUE	TRUE	FALSE	MAX. count OF cycles OF retry
	sbModePos		: BOOL;				//0	Non-RETAIN	TRUE	TRUE	TRUE	FALSE	Mode OF setting okay
	sxSendBuf		: sxSendBuf;		//	Non-RETAIN	TRUE	TRUE	TRUE	FALSE	send buffer OF telegram FOR sending data TO the drive
	sxRecvBuf		: sxRecvBuf;		//	Non-RETAIN	TRUE	TRUE	TRUE	FALSE	receive buffer OF telegram FOR receiving data FROM the drive

	piRetSFC	: INT;					//						Status FOR fault analysis
	piCount		: INT;					//						Freely available counter variable 3
	swSendBuf	: ARRAY[0..11] OF WORD;	//							Send buffer
	swRecvBuf	: ARRAY[0..11] OF WORD;	//							Receive buffer
	DPWR_DAT	: INT;
END_VAR


IF xLicensaValida5154156 THEN
	//=============================================================================
	//SIEMENS AG
	//(c)Copyright 2017 All Rights Reserved
	//-----------------------------------------------------------------------------
	// Library: DriveLib
	// Tested with: S7-1516-3 PN/DP V1.8
	// Engineering: TIA Portal V14
	// Restrictions: -
	// Requirements: S7-1200 / S7-1500
	// Functionality: cyclic communication between a SINAMICS (Basic positioner)and a PLC
	//                If in HWConfig Std.TLG 111 is projected 12 PZD-words are exchanged
	//                in every bus cycle.
	//                The parametrisation of these words is described in the manual of the
	//                SINAMICS
	// Trasferido para Beckhoff por Ricardo Gajardo e Tiago B. Cunico em 26/06/2021
	//=============================================================================
	
	// Betriebsart ermitteln
	IF ModePos > siModePosMax THEN
		sbModePos	:= FALSE;
		Error		:= TRUE;
		swStatus	:= 16#8202;
	ELSIF ModePos < 1 THEN
	
		sbModePos	:= FALSE;
		Error		:= TRUE;
		swStatus	:= 16#8202;
	ELSE
		// Betriebsartenwechsel ist nur möglich, wenn die Achse nicht beschleunigt oder nicht verzögert 
		// und die Geschwindigkeit Null ist
		IF NOT sbFWD AND NOT sbBWD AND NOT sbAccel AND NOT sbDecel THEN
	
			sbModePos	:= TRUE;
			siModePos	:= ModePos;
	
			// Fehler wieder zurücknehmen, wenn er mal ausgelöst wurde
			IF swStatus = 16#8202 THEN
				swStatus	:= 16#7002;
				Error		:= False;
			END_IF;
		END_IF;
	END_IF;
	
	// Überprüfung der analogen Eingabewerte, ob sie innerhalb des möglichen Bereiches liegen
	// Geschwindigkeitsoverride (0% - 199%, 100% => W16#4000)
	IF (OverV < 0) OR (OverV > 199) THEN
		swStatus	:= 16#8203;
		Error		:= True;
	ELSE
		// Geschwindigkeitsoverride in den Sendepuffer eintragen
		sxSendBuf.OverrideV := INT_TO_WORD(REAL_TO_INT(16384.0 * (INT_TO_REAL(OverV) / 100.0)));
	END_IF;
	
	// Beschleunigungsoverride (0% - 100%, 100% => W16#4000)
	IF (OverAcc < 0) OR (OverAcc > 100) THEN
		swStatus	:= 16#8203;
		Error		:= True;
	ELSE
		// Beschleunigungsoverride in den Sendepuffer eintragen
		sxSendBuf.OverrideA := INT_TO_WORD(REAL_TO_INT(16384.0 * (INT_TO_REAL(OverAcc) / 100.0)));
	END_IF;
	
	// Verzögerungsoverride (0% - 100%, 100% => W16#4000)
	IF (OverDec < 0) OR (OverDec > 100) THEN
		swStatus	:= 16#8203;
		Error		:= True;
	ELSE
		// Verzögerungsoverride in den Sendepuffer eintragen
		sxSendBuf.OverrideD := INT_TO_WORD(REAL_TO_INT(16384.0 * (INT_TO_REAL(OverDec) / 100.0)));
	END_IF;
	
	// Fehler wieder zurücknehmen, wenn er mal ausgelöst wurde
	IF NOT (OverV < 0) AND NOT (OverV > 199) AND NOT (OverAcc < 0) AND NOT (OverAcc > 100) AND NOT (OverDec < 0) AND NOT (OverDec > 100) THEN
		IF swStatus = 16#8203 THEN
			swStatus	:= 16#7002;
			Error		:= False;
		END_IF;
	END_IF;
	
	// Positionssollwert
	// Positionssollwert in den Sendepuffer eintragen
	sxSendBuf.Position.Valor := DINT_TO_DWORD(Position);
	
	// Geschwindigkeitssollwert (Begrenzung / Überwachung
	// Geschwindigkeitssollwert in den Sendepuffer eintragen
	sxSendBuf.Velocity.Valor := DINT_TO_DWORD(Velocity);
	
	// Einschalten bzw. Ausschalten des Antriebes erkennen
	IF EnableAxis AND NOT sbOff1Edge AND NOT sbBusy AND sbModePos THEN
		sbOff1 := True;
	END_IF;
	// Einschalten bzw. Ausschalten des Antriebes Flanke merken
	sbOff1Edge := EnableAxis AND NOT sbBusy;
	
	// Einschaltflankenmerker wieder zurücksetzen
	IF NOT EnableAxis THEN
		sbOff1 := False;
	END_IF;
	
	// Fliegendes Referenzieren aktivieren erkennen
	IF FlyRef AND NOT sbRefTypEdge THEN
		sbRefTyp := True;
	END_IF;
	// Fliegendes Referenzieren aktivieren Flanke merken
	sbRefTypEdge := FlyRef;
	
	// Fliegendes Referenzieren Flankenmerker wieder zurücksetzen
	IF NOT FlyRef THEN
		sbRefTyp	:= False;
		siRefTypCyc	:= 0;
	END_IF;
	
	// Verfahrauftrag aktivieren erkennen
	IF ExecuteMode AND NOT sbExecuteEdge THEN
		sbExecute := True;
	END_IF;
	// Verfahrauftrag aktivieren Flanke merken
	sbExecuteEdge := ExecuteMode;
	
	// Verfahrauftragflankenmerker wieder zurücksetzen
	IF NOT ExecuteMode THEN
		sbExecute		:= False;
		siExecuteCyc	:= 0;
	END_IF;
	
	// Betriebsart MDI / Sollwertdirektvorgabe Flanke merken
	
	(*IF sxSendBuf.sxEPosSTW1.MdiStart AND NOT sbMdiStartEdge THEN
			  sbMdiStart := True;
		  END_IF;
		  // Betriebsart MDI / Sollwertdirektvorgabe Flanke merken
		  sbMdiStartEdge := sxSendBuf.sxEPosSTW1.MdiStart AND NOT Busy;*)
	
	// Verfahrauftragflankenmerker wieder zurücksetzen
	
	(*IF NOT sxSendBuf.sxEPosSTW1.MdiStart THEN
			  sbMdiStart := False;
			  siMdiStartCyc := 0;
		  END_IF;*)
	
	IF sxSendBuf.EPosSTW1.x16b.bBit15 AND NOT sbMdiStartEdge THEN
		sbMdiStart := True;
	END_IF;
	// Betriebsart MDI / Sollwertdirektvorgabe Flanke merken
	sbMdiStartEdge := sxSendBuf.EPosSTW1.x16b.bBit15 AND NOT sbBusy;
	
	// Verfahrauftragflankenmerker wieder zurücksetzen
	IF NOT sxSendBuf.EPosSTW1.x16b.bBit15 THEN
		sbMdiStart		:= False;
		siMdiStartCyc	:= 0;
	END_IF;
	
	// Schreibdaten zusammenstellen
	// Steuerword STW1 für alle Betriebsart aufbereiten
	
	(*sxSendBuf.sxSTW1.RejTrvTsk        := RejTrvTsk;
		  sxSendBuf.sxSTW1.IntMStop         := IntMStop;
		  sxSendBuf.sxSTW1.AckFault         := AckFlt;*)
	
	sxSendBuf.STW1.x16b.bBit4	:= CancelTraversing;
	sxSendBuf.STW1.x16b.bBit5	:= IntermediateStop;
	sxSendBuf.STW1.x16b.bBit7	:= AckError;
	sxSendBuf.STW1.x16b.bBit1	:= TRUE;
	sxSendBuf.STW1.x16b.bBit2	:= TRUE;
	sxSendBuf.STW1.x16b.bBit3	:= TRUE;
	sxSendBuf.STW1.x16b.bBit10	:= TRUE;
	
	// Hauptbetriebsart "Positionieren / manueller Sollwertvorgabe (MDI)" 
	// Betriebsart "Positionieren Relativ positiv" oder "Positionieren Relativ negativ"
	IF (siModePos = 1 AND sbModePos) THEN
	
		// Antrieb einschalten
		//sxSendBuf.sxSTW1.Off1 := sbOff1;
		sxSendBuf.STW1.x16b.bBit0 := sbOff1;
	
		// nicht verwendete Signale für den 1. Schritt und eventuell weitere Schritte
	
		(*sxSendBuf.sxSTW1.Jog1          := False;
			  sxSendBuf.sxSTW1.Jog2          := False;
			  sxSendBuf.sxEPosSTW1.MdiTyp    := False;
			  sxSendBuf.sxEPosSTW1.MdiPos    := False;
			  sxSendBuf.sxEPosSTW1.MdiNeg    := False;
			  sxSendBuf.sxEPosSTW1.MdiSetup  := False;
			  sxSendBuf.sxEPosSTW2.SetRefPt  := False;
			  sxSendBuf.sxEPosSTW2.JogInc    := False;
			  sxSendBuf.sxEPosSTW2.RefStDi   := False;
			  sxSendBuf.sxSTW1.RefStart      := False;
			  sxSendBuf.sxEPosSTW2.RefTyp    := False;
			  sxSendBuf.sxEPosSTW1.MdiStart  := False;*)
	
		sxSendBuf.STW1.x16b.bBit8		:= False;
		sxSendBuf.STW1.x16b.bBit9		:= False;
		sxSendBuf.EPosSTW1.x16b.bBit8	:= False;
		sxSendBuf.EPosSTW1.x16b.bBit9	:= False;
		sxSendBuf.EPosSTW1.x16b.bBit10	:= False;
		sxSendBuf.EPosSTW1.x16b.bBit14	:= False;
		sxSendBuf.EPosSTW2.x16b.bBit1	:= False;
		sxSendBuf.EPosSTW2.x16b.bBit5	:= False;
		sxSendBuf.EPosSTW2.x16b.bBit9	:= False;
		sxSendBuf.STW1.x16b.bBit11		:= False;
		sxSendBuf.EPosSTW2.x16b.bBit8	:= False;
		sxSendBuf.EPosSTW1.x16b.bBit15	:= False;
	
		// Nach dem Einschalten des Antriebes, prüfen ob der Antrieb betriebsbereit, in Operation ohne Fehler und Warnung ist, 
		// dann die Betriebsart MDI / Sollwertvorgabe Start gesetzt werden
		IF sbOff1 AND sbReady AND sbIOp AND NOT sbFault THEN
	
			// Betriebsart MDI / Sollwertdirektvorgabe setzen
			//sxSendBuf.sxEPosSTW1.MdiStart := True;
			sxSendBuf.EPosSTW1.x16b.bBit15 := True;
	
			// Positioniertyp auf relatives Positionieren stellen 
			//sxSendBuf.sxEPosSTW1.MdiTyp := False;
			sxSendBuf.EPosSTW1.x16b.bBit8 := False;
	
			// die Richtungswahl für das Positionieren auf positive Richtung oder negative Richtung einstellen
			IF Positive AND NOT Negative THEN
	
				// positive Richtung
				//sxSendBuf.sxEPosSTW1.MdiPos := True;
				sxSendBuf.EPosSTW1.x16b.bBit9 := True;
	
				// negative Richtung
				//sxSendBuf.sxEPosSTW1.MdiNeg := False;
				sxSendBuf.EPosSTW1.x16b.bBit10 := False;
	
				// die Richtungswahl für das Positionieren auf negative Richtung einstellen                
			ELSIF NOT Positive AND Negative THEN
	
				// positive Richtung
				//sxSendBuf.sxEPosSTW1.MdiPos := False;
				sxSendBuf.EPosSTW1.x16b.bBit9 := False;
	
				// negative Richtung
				//sxSendBuf.sxEPosSTW1.MdiNeg := True;
				sxSendBuf.EPosSTW1.x16b.bBit10 := True;
	
				// die Richtungswahl für das Positionieren auf keine Richtung einstellen                
			ELSE
	
				// positive Richtung
				//sxSendBuf.sxEPosSTW1.MdiPos := False;
				sxSendBuf.EPosSTW1.x16b.bBit9 := False;
	
				// negative Richtung
				//sxSendBuf.sxEPosSTW1.MdiNeg := False;
				sxSendBuf.EPosSTW1.x16b.bBit10 := False;
	
			END_IF;
	
			// Nach dem Einschalten des Antriebes und dem Betriebsart MDI / Sollwertvorgabe starten, 
			// ein Paar Zyklen warten bevor die Flanke für die Sollwertübernahme MDI gesetzt werden kann
			IF sbMdiStart AND (siMdiStartCyc < siCycWait) THEN
				siMdiStartCyc := siMdiStartCyc + 1;
			ELSE
				// Flanke Sollwertübernahme MDI
				//sxSendBuf.sxSTW1.TrvStart := Execute;
				sxSendBuf.STW1.x16b.bBit6 := ExecuteMode;
	
			END_IF;
	
			// "Fliegendes Referentieren" aktivieren
			// "Fliegendes Referenzieren" erst nach Einschalten des Antriebes möglich
			IF sbRefTyp THEN
	
				// Referenziertyp auf "Fliegendes Referenzieren" einstellen
				//sxSendBuf.sxEPosSTW2.RefTyp := True;
				sxSendBuf.EPosSTW2.x16b.bBit8 := True;
	
				// Nach der Anwahl des Referenziertyps "Fliegendes Referenzieren", 
				// ein Zyklus später kann das Referenzieren gestartet
				IF (siRefTypCyc = 0) THEN
					siRefTypCyc := siRefTypCyc + 1;
				ELSE
					// Referenzieren starten
					//sxSendBuf.sxSTW1.RefStart := True;
					sxSendBuf.STW1.x16b.bBit11 := True;
	
				END_IF;
			END_IF;
		END_IF;
	
		// Betriebsart "Positionieren Absolut" oder "Positonieren Absolut positiv" oder "Positionieren Absolut negativ"
	ELSIF siModePos = 2 AND sbModePos THEN
	
		// Antrieb einschalten
		//sxSendBuf.sxSTW1.Off1 := sbOff1;
		sxSendBuf.STW1.x16b.bBit0 := sbOff1;
	
		// nicht verwendete Signale für den 1. Schritt und eventuell weitere Schritte
	
		(*sxSendBuf.sxSTW1.Jog1         := False;
			  sxSendBuf.sxSTW1.Jog2         := False;
			  sxSendBuf.sxEPosSTW1.MdiTyp   := False;
			  sxSendBuf.sxEPosSTW1.MdiPos   := False;
			  sxSendBuf.sxEPosSTW1.MdiNeg   := False;
			  sxSendBuf.sxEPosSTW1.MdiSetup := False;
			  sxSendBuf.sxEPosSTW2.SetRefPt := False;
			  sxSendBuf.sxEPosSTW2.JogInc   := False;
			  sxSendBuf.sxEPosSTW2.RefStDi  := False;
			  sxSendBuf.sxSTW1.RefStart     := False;
			  sxSendBuf.sxEPosSTW2.RefTyp   := False;
			  sxSendBuf.sxEPosSTW1.MdiStart := False;*)
	
		sxSendBuf.STW1.x16b.bBit8		:= False;
		sxSendBuf.STW1.x16b.bBit9		:= False;
		sxSendBuf.EPosSTW1.x16b.bBit8	:= False;
		sxSendBuf.EPosSTW1.x16b.bBit9	:= False;
		sxSendBuf.EPosSTW1.x16b.bBit10	:= False;
		sxSendBuf.EPosSTW1.x16b.bBit14	:= False;
		sxSendBuf.EPosSTW2.x16b.bBit1	:= False;
		sxSendBuf.EPosSTW2.x16b.bBit5	:= False;
		sxSendBuf.EPosSTW2.x16b.bBit9	:= False;
		sxSendBuf.STW1.x16b.bBit11		:= False;
		sxSendBuf.EPosSTW2.x16b.bBit8	:= False;
		sxSendBuf.EPosSTW1.x16b.bBit15	:= False;
	
		// Nach dem Einschalten des Antriebes, prüfen ob der Antrieb betriebsbereit, in Operation ohne Fehler und Warnung ist, 
		// dann die Betriebsart MDI / Sollwertvorgabe Start gesetzt werden
		IF sbOff1 AND sbReady AND sbIOp AND NOT sbFault THEN
	
			// Betriebsart MDI / Sollwertdirektvorgabe setzen
			//sxSendBuf.sxEPosSTW1.MdiStart := True;
			sxSendBuf.EPosSTW1.x16b.bBit15 := True;
	
			// Positioniertyp auf absolutes Positionieren stellen 
			//sxSendBuf.sxEPosSTW1.MdiTyp := True;
			sxSendBuf.EPosSTW1.x16b.bBit8 := True;
	
			// die Richtungswahl für das Positionieren auf positive Richtung oder negative Richtung einstellen
			IF Positive AND NOT Negative THEN
	
				// positive Richtung
				//sxSendBuf.sxEPosSTW1.MdiPos := True;
				sxSendBuf.EPosSTW1.x16b.bBit9 := True;
	
				// negative Richtung
				//sxSendBuf.sxEPosSTW1.MdiNeg := False;
				sxSendBuf.EPosSTW1.x16b.bBit10 := False;
	
				// die Richtungswahl für das Positionieren auf negative Richtung einstellen                
			ELSIF NOT Positive AND Negative THEN
	
				// positive Richtung
				//sxSendBuf.sxEPosSTW1.MdiPos := False;
				sxSendBuf.EPosSTW1.x16b.bBit9 := False;
	
				// negative Richtung
				//sxSendBuf.sxEPosSTW1.MdiNeg := True;
				sxSendBuf.EPosSTW1.x16b.bBit10 := True;
	
				// die Richtungswahl für das Positionieren auf keine Richtung einstellen                
			ELSE
	
				// positive Richtung
				//sxSendBuf.sxEPosSTW1.MdiPos := False;
				sxSendBuf.EPosSTW1.x16b.bBit9 := False;
	
				// negative Richtung
				//sxSendBuf.sxEPosSTW1.MdiNeg := False;
				sxSendBuf.EPosSTW1.x16b.bBit10 := False;
	
			END_IF;
	
			// Nach dem Einschalten des Antriebes und dem Betriebsart MDI / Sollwertvorgabe starten, 
			// ein Paar Zyklen warten bevor die Flanke für die Sollwertübernahme MDI gesetzt werden kann
			IF sbMdiStart AND (siMdiStartCyc < siCycWait) THEN
				siMdiStartCyc := siMdiStartCyc + 1;
			ELSE
				// Flanke Sollwertübernahme MDI
				//sxSendBuf.sxSTW1.TrvStart := Execute;
				sxSendBuf.STW1.x16b.bBit6 := ExecuteMode;
	
			END_IF;
	
			// "Fliegendes Referentieren" aktivieren
			// "Fliegendes Referenzieren" erst nach Einschalten des Antriebes möglich
			IF sbRefTyp THEN
	
				// Referenziertyp auf "Fliegendes Referenzieren" einstellen
				//sxSendBuf.sxEPosSTW2.RefTyp := True;
				sxSendBuf.EPosSTW2.x16b.bBit8 := True;
	
				// Nach der Anwahl des Referenziertyps "Fliegendes Referenzieren", 
				// ein Zyklus später kann das Referenzieren gestartet
				IF (siRefTypCyc = 0) THEN
					siRefTypCyc := siRefTypCyc + 1;
				ELSE
					// Referenzieren starten
					//sxSendBuf.sxSTW1.RefStart := True;
					sxSendBuf.STW1.x16b.bBit11 := True;
	
				END_IF;
			END_IF;
		END_IF;
	
		// Betriebsart "Positionieren als Einrichten positiv" oder "Positionieren als Einrichten negativ"
	ELSIF siModePos = 3 AND sbModePos THEN
	
		// Antrieb einschalten
		//sxSendBuf.sxSTW1.Off1 := sbOff1;
		sxSendBuf.STW1.x16b.bBit0 := sbOff1;
	
		// nicht verwendete Signale für den 1. Schritt und eventuell weitere Schritte
	
		(*sxSendBuf.sxSTW1.Jog1           := False;
			  sxSendBuf.sxSTW1.Jog2           := False;
			  sxSendBuf.sxEPosSTW1.MdiTyp     := False;
			  sxSendBuf.sxEPosSTW1.MdiPos     := False;
			  sxSendBuf.sxEPosSTW1.MdiNeg     := False;
			  sxSendBuf.sxEPosSTW1.MdiSetup   := False;
			  sxSendBuf.sxEPosSTW2.SetRefPt   := False;
			  sxSendBuf.sxEPosSTW2.JogInc     := False;
			  sxSendBuf.sxEPosSTW2.RefStDi    := False;
			  sxSendBuf.sxSTW1.RefStart       := False;
			  sxSendBuf.sxEPosSTW2.RefTyp     := False;
			  sxSendBuf.sxEPosSTW1.MdiStart   := False;*)
	
		sxSendBuf.STW1.x16b.bBit8		:= False;
		sxSendBuf.STW1.x16b.bBit9		:= False;
		sxSendBuf.EPosSTW1.x16b.bBit8	:= False;
		sxSendBuf.EPosSTW1.x16b.bBit9	:= False;
		sxSendBuf.EPosSTW1.x16b.bBit10	:= False;
		sxSendBuf.EPosSTW1.x16b.bBit14	:= False;
		sxSendBuf.EPosSTW2.x16b.bBit1	:= False;
		sxSendBuf.EPosSTW2.x16b.bBit5	:= False;
		sxSendBuf.EPosSTW2.x16b.bBit9	:= False;
		sxSendBuf.STW1.x16b.bBit11		:= False;
		sxSendBuf.EPosSTW2.x16b.bBit8	:= False;
		sxSendBuf.EPosSTW1.x16b.bBit15	:= False;
	
		// Nach dem Einschalten des Antriebes, prüfen ob der Antrieb betriebsbereit, in Operation ohne Fehler und Warnung ist, 
		// dann die Betriebsart MDI / Sollwertvorgabe Start gesetzt werden
		IF sbOff1 AND sbReady AND sbIOp AND NOT sbFault THEN
	
			// Betriebsart MDI / Sollwertdirektvorgabe setzen
			//sxSendBuf.sxEPosSTW1.MdiStart := True;
			sxSendBuf.EPosSTW1.x16b.bBit15 := True;
	
			// Positioniertyp auf absolutes Positionieren stellen 
			//sxSendBuf.sxEPosSTW1.MdiTyp := True;
			sxSendBuf.EPosSTW1.x16b.bBit8 := True;
	
			// die Anwahl für MDI Modus auf Einrichten einstellen
			//sxSendBuf.sxEPosSTW1.MdiSetup := True;
			sxSendBuf.EPosSTW1.x16b.bBit14 := True;
	
			// die Richtungswahl für das Positionieren auf positive Richtung oder negative Richtung einstellen
			IF Positive AND NOT Negative THEN
	
				// positive Richtung
				//sxSendBuf.sxEPosSTW1.MdiPos := True;
				sxSendBuf.EPosSTW1.x16b.bBit9 := True;
	
				// negative Richtung
				//sxSendBuf.sxEPosSTW1.MdiNeg := False;
				sxSendBuf.EPosSTW1.x16b.bBit10 := False;
	
				// die Richtungswahl für das Positionieren auf negative Richtung einstellen                
			ELSIF NOT Positive AND Negative THEN
	
				// positive Richtung
				//sxSendBuf.sxEPosSTW1.MdiPos := False;
				sxSendBuf.EPosSTW1.x16b.bBit9 := False;
	
				// negative Richtung
				//sxSendBuf.sxEPosSTW1.MdiNeg := True;
				sxSendBuf.EPosSTW1.x16b.bBit10 := True;
	
				// die Richtungswahl für das Positionieren auf keine Richtung einstellen                
			ELSE
	
				// positive Richtung
				//sxSendBuf.sxEPosSTW1.MdiPos := False;
				sxSendBuf.EPosSTW1.x16b.bBit9 := False;
	
				// negative Richtung
				//sxSendBuf.sxEPosSTW1.MdiNeg := False;
				sxSendBuf.EPosSTW1.x16b.bBit10 := False;
	
			END_IF;
	
			// Nach dem Einschalten des Antriebes und dem Betriebsart MDI / Sollwertvorgabe starten, 
			// ein Paar Zyklen warten bevor die Flanke für die Sollwertübernahme MDI gesetzt werden kann
			IF sbMdiStart AND (siMdiStartCyc < siCycWait) THEN
				siMdiStartCyc := siMdiStartCyc + 1;
			ELSE
				// Flanke Sollwertübernahme MDI
				//sxSendBuf.sxSTW1.TrvStart := Execute;
				sxSendBuf.STW1.x16b.bBit6 := ExecuteMode;
	
			END_IF;
	
			// "Fliegendes Referentieren" aktivieren
			// "Fliegendes Referenzieren" erst nach Einschalten des Antriebes möglich
			IF sbRefTyp THEN
	
				// Referenziertyp auf "Fliegendes Referenzieren" einstellen
				//sxSendBuf.sxEPosSTW2.RefTyp := True;
				sxSendBuf.EPosSTW2.x16b.bBit8 := True;
	
				// Nach der Anwahl des Referenziertyps "Fliegendes Referenzieren", 
				// ein Zyklus später kann das Referenzieren gestartet
				IF (siRefTypCyc = 0) THEN
					siRefTypCyc := siRefTypCyc + 1;
				ELSE
					// Referenzieren starten
					//sxSendBuf.sxSTW1.RefStart := True;
					sxSendBuf.STW1.x16b.bBit11 := True;
	
				END_IF;
			END_IF;
		END_IF;
	
		// Hauptbetriebsart "Referenzieren" (Reference)
		// Betriebsart "Referenzieren - Referenzpunktfahrt positiv" oder "Referenzieren - Referenzpunktfahrt negativ"
	ELSIF siModePos = 4 AND sbModePos THEN
	
		// Antrieb einschalten
		//sxSendBuf.sxSTW1.Off1 := sbOff1;
		sxSendBuf.STW1.x16b.bBit0 := sbOff1;
	
		// nicht verwendete Signale für den 1. Schritt und eventuell weitere Schritte
	
		(*sxSendBuf.sxSTW1.Jog1         := False;
			  sxSendBuf.sxSTW1.Jog2         := False;
			  sxSendBuf.sxEPosSTW1.MdiStart := False;
			  sxSendBuf.sxEPosSTW2.SetRefPt := False;
			  sxSendBuf.sxEPosSTW2.JogInc   := False;
			  sxSendBuf.sxEPosSTW2.RefTyp   := False;
			  sxSendBuf.sxSTW1.RefStart     := False;
			  sxSendBuf.sxEPosSTW2.RefStDi  := False;*)
	
		sxSendBuf.STW1.x16b.bBit8		:= False;
		sxSendBuf.STW1.x16b.bBit9		:= False;
		sxSendBuf.EPosSTW1.x16b.bBit15	:= False;
		sxSendBuf.EPosSTW2.x16b.bBit1	:= False;
		sxSendBuf.EPosSTW2.x16b.bBit5	:= False;
		sxSendBuf.EPosSTW2.x16b.bBit8	:= False;
		sxSendBuf.STW1.x16b.bBit11		:= False;
		sxSendBuf.EPosSTW2.x16b.bBit9	:= False;
	
		// Nach dem Einschalten des Antriebes, prüfen ob der Antrieb betriebsbereit, in Operation ohne Fehler und Warnung ist, 
		// dann die Betriebsart MDI / Sollwertvorgabe Start gesetzt werden
		IF sbOff1 AND sbReady AND sbIOp AND NOT sbFault THEN
	
			// Referenzieren starten
			//sxSendBuf.sxSTW1.RefStart := Execute;
			sxSendBuf.STW1.x16b.bBit11 := ExecuteMode;
	
			// die Richtungswahl für das Referenzpunktfahrt positiv einstellen
			IF Positive AND NOT Negative THEN
	
				// positive Referenzpunktfahrt
				//sxSendBuf.sxEPosSTW2.RefStDi := False;
				sxSendBuf.EPosSTW2.x16b.bBit9 := False;
	
				// die Richtungswahl für das Referenzpunktfahrt negativ einstellen                
			ELSIF NOT Positive AND Negative THEN
	
				// negative Referenzpunktfahrt
				//sxSendBuf.sxEPosSTW2.RefStDi := True;
				sxSendBuf.EPosSTW2.x16b.bBit9 := True;
	
			END_IF;
		END_IF;
	
		// Betriebsart "Referenzieren - Referenzpunkt setzen"
	ELSIF siModePos = 5 AND sbModePos THEN
	
		// Antrieb einschalten
		//sxSendBuf.sxSTW1.Off1 := sbOff1;
		sxSendBuf.STW1.x16b.bBit0 := sbOff1;
	
		// nicht verwendete Signale für den 1. Schritt und eventuell weitere Schritte
	
		(*sxSendBuf.sxSTW1.Jog1          := False;
			  sxSendBuf.sxSTW1.Jog2          := False;
			  sxSendBuf.sxSTW1.RefStart      := False;
			  sxSendBuf.sxEPosSTW1.MdiStart  := False;
			  sxSendBuf.sxEPosSTW2.JogInc    := False;
			  sxSendBuf.sxEPosSTW2.RefTyp    := False;
			  sxSendBuf.sxEPosSTW2.RefStDi   := False;
			  sxSendBuf.sxEPosSTW2.SetRefPt  := False;*)
	
		sxSendBuf.STW1.x16b.bBit8		:= False;
		sxSendBuf.STW1.x16b.bBit9		:= False;
		sxSendBuf.STW1.x16b.bBit11		:= False;
		sxSendBuf.EPosSTW1.x16b.bBit15	:= False;
		sxSendBuf.EPosSTW2.x16b.bBit5	:= False;
		sxSendBuf.EPosSTW2.x16b.bBit8	:= False;
		sxSendBuf.EPosSTW2.x16b.bBit9	:= False;
		sxSendBuf.EPosSTW2.x16b.bBit1	:= False;
	
		// Nach dem Einschalten des Antriebes, prüfen ob der Antrieb betriebsbereit, in Operation ohne Fehler und Warnung ist, 
		// dann die Betriebsart MDI / Sollwertvorgabe Start gesetzt werden
		IF NOT sbFault THEN
	
			// Referenzpunktfahrt negativ
			//sxSendBuf.sxEPosSTW2.SetRefPt := Execute;
			sxSendBuf.EPosSTW2.x16b.bBit1 := ExecuteMode;
	
		END_IF;
	
		// Hauptbetriebsart "Verfahrsätze" (Traversing Blocks)
	ELSIF siModePos = 6 AND sbModePos THEN
	
		// Antrieb einschalten
		//sxSendBuf.sxSTW1.Off1 := sbOff1;
		sxSendBuf.STW1.x16b.bBit0 := sbOff1;
	
		// nicht verwendete Signale für den 1. Schritt und eventuell weitere Schritte
	
		(*sxSendBuf.sxSTW1.Jog1          := False;
			  sxSendBuf.sxSTW1.Jog2          := False;
			  sxSendBuf.sxEPosSTW1.MdiTyp    := False;
			  sxSendBuf.sxEPosSTW1.MdiPos    := False;
			  sxSendBuf.sxEPosSTW1.MdiNeg    := False;
			  sxSendBuf.sxEPosSTW1.MdiSetup  := False;
			  sxSendBuf.sxEPosSTW2.SetRefPt  := False;
			  sxSendBuf.sxEPosSTW2.JogInc    := False;
			  sxSendBuf.sxEPosSTW2.RefStDi   := False;
			  sxSendBuf.sxEPosSTW2.RefTyp    := False;
			  sxSendBuf.sxSTW1.RefStart      := False;
			  sxSendBuf.sxEPosSTW1.TrvBit0   := False;
			  sxSendBuf.sxEPosSTW1.TrvBit1   := False;
			  sxSendBuf.sxEPosSTW1.TrvBit2   := False;
			  sxSendBuf.sxEPosSTW1.TrvBit3   := False;
			  sxSendBuf.sxEPosSTW1.TrvBit4   := False;
			  sxSendBuf.sxEPosSTW1.TrvBit5   := False;
			  sxSendBuf.sxEPosSTW1.MdiStart  := False;*)
	
		sxSendBuf.STW1.x16b.bBit8		:= False;
		sxSendBuf.STW1.x16b.bBit9		:= False;
		sxSendBuf.EPosSTW1.x16b.bBit8	:= False;
		sxSendBuf.EPosSTW1.x16b.bBit9	:= False;
		sxSendBuf.EPosSTW1.x16b.bBit10	:= False;
		sxSendBuf.EPosSTW1.x16b.bBit14	:= False;
		sxSendBuf.EPosSTW2.x16b.bBit1	:= False;
		sxSendBuf.EPosSTW2.x16b.bBit5	:= False;
		sxSendBuf.EPosSTW2.x16b.bBit9	:= False;
		sxSendBuf.EPosSTW2.x16b.bBit8	:= False;
		sxSendBuf.STW1.x16b.bBit11		:= False;
		sxSendBuf.EPosSTW1.x16b.bBit0	:= False;
		sxSendBuf.EPosSTW1.x16b.bBit1	:= False;
		sxSendBuf.EPosSTW1.x16b.bBit2	:= False;
		sxSendBuf.EPosSTW1.x16b.bBit3	:= False;
		sxSendBuf.EPosSTW1.x16b.bBit4	:= False;
		sxSendBuf.EPosSTW1.x16b.bBit5	:= False;
		sxSendBuf.EPosSTW1.x16b.bBit15	:= False;
	
		// Bei der Auswahl der Verfahrsätze entspricht die Position der Verfahrensatznummer 
		// Verfahrsatznummer aus der Position ermitteln und in die einzelnen Bit's aufteilen
		// Es sind die Verfahrsatznummern 0 - 63 möglich
		IF (DINT_TO_INT(Position) < 0) OR (DINT_TO_INT(Position) > 63) THEN
			// Fehler, ungültiger Verfahrsatznummer
			swStatus	:= 16#8204;
			Error		:= True;
		ELSE
			// Fehler wieder zurücknehmen, wenn er mal ausgelöst wurde
			IF swStatus = 16#8204 THEN
				swStatus	:= 16#7002;
				Error		:= False;
			END_IF;
	
			// Verfahrsatznummer Bit 0 ermitteln
			IF (DINT_TO_WORD(Position) AND 16#01) = 16#01 THEN
				//sxSendBuf.sxEPosSTW1.TrvBit0 := True;
				sxSendBuf.EPosSTW1.x16b.bBit0 := True;
			END_IF;
	
			// Verfahrsatznummer Bit 1 ermitteln
			IF (DINT_TO_WORD(Position) AND 16#02) = 16#02 THEN
				//sxSendBuf.sxEPosSTW1.TrvBit1 := True;
				sxSendBuf.EPosSTW1.x16b.bBit1 := True;
			END_IF;
	
			// Verfahrsatznummer Bit 2 ermitteln
			IF (DINT_TO_WORD(Position) AND 16#04) = 16#04 THEN
				//sxSendBuf.sxEPosSTW1.TrvBit2 := True;
				sxSendBuf.EPosSTW1.x16b.bBit2 := True;
			END_IF;
	
			// Verfahrsatznummer Bit 3 ermitteln
			IF (DINT_TO_WORD(Position) AND 16#08) = 16#08 THEN
				//sxSendBuf.sxEPosSTW1.TrvBit3 := True;
				sxSendBuf.EPosSTW1.x16b.bBit3 := True;
			END_IF;
	
			// Verfahrsatznummer Bit 4 ermitteln
			IF (DINT_TO_WORD(Position) AND 16#10) = 16#10 THEN
				//sxSendBuf.sxEPosSTW1.TrvBit4 := True;
				sxSendBuf.EPosSTW1.x16b.bBit4 := True;
			END_IF;
	
			// Verfahrsatznummer Bit 5 ermitteln
			IF (DINT_TO_WORD(Position) AND 16#20) = 16#20 THEN
				//sxSendBuf.sxEPosSTW1.TrvBit5 := True;
				sxSendBuf.EPosSTW1.x16b.bBit5 := True;
			END_IF;
	
			// Nach dem Einschalten des Antriebes, prüfen ob der Antrieb betriebsbereit, in Operation ohne Fehler und Warnung ist, 
			// dann die Betriebsart MDI / Sollwertvorgabe Start gesetzt werden
			IF sbOff1 AND sbReady AND sbIOp AND NOT sbFault THEN
	
				// Positioniertyp auf absolutes Positionieren stellen 
				//sxSendBuf.sxEPosSTW1.MdiTyp := True;
				sxSendBuf.EPosSTW1.x16b.bBit8 := True;
	
				// die Richtungswahl für das Positionieren auf positive Richtung einstellen
				//sxSendBuf.sxEPosSTW1.MdiPos := True;
				sxSendBuf.EPosSTW1.x16b.bBit9 := True;
	
				// die Richtungswahl für das Positionieren auf negative Richtung abstellen
				//sxSendBuf.sxEPosSTW1.MdiNeg := False;
				sxSendBuf.EPosSTW1.x16b.bBit10 := False;
	
				// die Anwahl für MDI Modus auf Einrichten einstellen
				//sxSendBuf.sxEPosSTW1.MdiSetup := True;
				sxSendBuf.EPosSTW1.x16b.bBit14 := True;
	
				// Nach dem Einschalten des Antriebes und dem Betriebsart MDI / Sollwertvorgabe starten, 
				// ein Paar Zyklen warten bevor die Flanke für die Sollwertübernahme MDI gesetzt werden kann
				IF sbMdiStart AND (siMdiStartCyc < siCycWait) THEN
					siMdiStartCyc := siMdiStartCyc + 1;
				ELSE
					// Flanke Sollwertübernahme MDI
					//sxSendBuf.sxSTW1.TrvStart := Execute;
					sxSendBuf.STW1.x16b.bBit6 := ExecuteMode;
				END_IF;
	
				// "Fliegendes Referentieren" aktivieren
				// "Fliegendes Referenzieren" erst nach Einschalten des Antriebes möglich
				IF sbRefTyp THEN
	
					// Referenziertyp auf "Fliegendes Referenzieren" einstellen
					//sxSendBuf.sxEPosSTW2.RefTyp := True;
					sxSendBuf.EPosSTW2.x16b.bBit8 := True;
	
					// Nach der Anwahl des Referenziertyps "Fliegendes Referenzieren", 
					// ein Zyklus später kann das Referenzieren gestartet
					IF (siRefTypCyc = 0) THEN
						siRefTypCyc := siRefTypCyc + 1;
					ELSE
						// Referenzieren starten
						//sxSendBuf.sxSTW1.RefStart := True;
						sxSendBuf.STW1.x16b.bBit11 := True;
					END_IF;
				END_IF;
			END_IF;
		END_IF;
	
		// Hauptbetriebsart "Tippen" (Jogging)
		// Betriebsart "Tippen positiv" oder "Tippen negativ" angewählt 
	ELSIF siModePos = 7 AND sbModePos THEN
	
		// Antrieb einschalten
		//sxSendBuf.sxSTW1.Off1 := sbOff1;
		sxSendBuf.STW1.x16b.bBit0 := sbOff1;
	
		// nicht verwendete Signale für den 1. Schritt und eventuell weitere Schritte
	
		(*sxSendBuf.sxEPosSTW1.MdiStart := False;
			  sxSendBuf.sxEPosSTW2.JogInc   := False;
			  sxSendBuf.sxSTW1.Jog1         := False;
			  sxSendBuf.sxSTW1.Jog2         := False;
			  sxSendBuf.sxEPosSTW2.RefTyp   := False;
			  sxSendBuf.sxSTW1.RefStart     := False;*)
	
		sxSendBuf.EPosSTW1.x16b.bBit15	:= False;
		sxSendBuf.EPosSTW2.x16b.bBit5	:= False;
		sxSendBuf.STW1.x16b.bBit8		:= False;
		sxSendBuf.STW1.x16b.bBit9		:= False;
		sxSendBuf.EPosSTW2.x16b.bBit8	:= False;
		sxSendBuf.STW1.x16b.bBit11		:= False;
	
		// Nach dem Einschalten des Antriebes, prüfen ob der Antrieb betriebsbereit, in Operation ohne Fehler und Warnung ist, 
		// dann kann Tippen positiv oder negativ gesetzt werden
		IF sbOff1 AND sbReady AND sbIOp AND NOT sbFault THEN
	
			// Tippen positiv
			IF Jog1 AND NOT Jog2 THEN
				//sxSendBuf.sxSTW1.Jog1 := True;
				sxSendBuf.STW1.x16b.bBit8 := True;
			END_IF;
	
			// Tippen negativ
			IF Jog2 AND NOT Jog1 THEN
				//sxSendBuf.sxSTW1.Jog2 := True;
				sxSendBuf.STW1.x16b.bBit9 := True;
			END_IF;
	
			// "Fliegendes Referentieren" aktivieren
			// "Fliegendes Referenzieren" erst nach Einschalten des Antriebes möglich
			IF sbRefTyp THEN
	
				// Referenziertyp auf "Fliegendes Referenzieren" einstellen
				//sxSendBuf.sxEPosSTW2.RefTyp := FlyRef;
				sxSendBuf.EPosSTW2.x16b.bBit8 := FlyRef;
	
				// Nach der Anwahl des Referenziertyps "Fliegendes Referenzieren", 
				// ein Zyklus später kann das Referenzieren gestartet
				IF (siRefTypCyc = 0) THEN
					siRefTypCyc := siRefTypCyc + 1;
				ELSE
					// Referenzieren starten
					//sxSendBuf.sxSTW1.RefStart := True;
					sxSendBuf.STW1.x16b.bBit11 := True;
				END_IF;
			END_IF;
		END_IF;
	
		// Betriebsart "Tippen positiv / Tippen negativ inkrementell" 
	ELSIF siModePos = 8 AND sbModePos THEN
	
		// Antrieb einschalten
		//sxSendBuf.sxSTW1.OFF1 := sbOff1;
		sxSendBuf.STW1.x16b.bBit0 := sbOff1;
	
		// nicht verwendete Signale für den 1. Schritt und eventuell weitere Schritte
	
		(*sxSendBuf.sxEPosSTW1.MdiStart := False;
			  sxSendBuf.sxEPosSTW2.JogInc   := False;
			  sxSendBuf.sxSTW1.Jog1         := False;
			  sxSendBuf.sxSTW1.Jog2         := False;
			  sxSendBuf.sxSTW1.RefStart     := False;
			  sxSendBuf.sxEPosSTW2.RefTyp   := False;*)
	
		sxSendBuf.EPosSTW1.x16b.bBit15	:= False;
		sxSendBuf.EPosSTW2.x16b.bBit5	:= False;
		sxSendBuf.STW1.x16b.bBit8		:= False;
		sxSendBuf.STW1.x16b.bBit9		:= False;
		sxSendBuf.STW1.x16b.bBit11		:= False;
		sxSendBuf.EPosSTW2.x16b.bBit8	:= False;
	
		// Nach dem Einschalten des Antriebes, ein Paar Zyklen warten bevor Tippen negativ gesetzt werden kann
		// Nach dem Einschalten des Antriebes, prüfen ob der Antrieb betriebsbereit, in Operation ohne Fehler und Warnung ist, 
		// dann kann Tippen positiv oder negativ gesetzt werden
		IF sbOff1 AND sbReady AND sbIOp AND NOT sbFault THEN
	
			// Tippen inkrementell einstellen
			//sxSendBuf.sxEPosSTW2.JogInc := True;
			sxSendBuf.EPosSTW2.x16b.bBit5 := True;
	
			sbJogInc := True;
	
			// Nach dem Einstellen des Antriebes, ein Paar Zyklen warten bevor Tippen negativ oder Tippen positiv gesetz werden kann
			IF sbJogInc AND (siJogIncCyc = 0) THEN
				siJogIncCyc := siJogIncCyc + 1;
			ELSE
	
				// Tippen positiv oder negativ inkrementell zulassen
				IF Jog1 XOR Jog2 THEN
	
					//sxSendBuf.sxSTW1.Jog1 := Jog1;
					//sxSendBuf.sxSTW1.Jog2 := Jog2;
					sxSendBuf.STW1.x16b.bBit8	:= Jog1;
					sxSendBuf.STW1.x16b.bBit9	:= Jog2;
				END_IF;
			END_IF;
	
			// "Fliegendes Referentieren" aktivieren
			// "Fliegendes Referenzieren" erst nach Einschalten des Antriebes möglich
			IF sbRefTyp THEN
	
				// Referenziertyp auf "Fliegendes Referenzieren" einstellen
				//sxSendBuf.sxEPosSTW2.RefTyp := True;
				sxSendBuf.EPosSTW2.x16b.bBit8 := True;
	
				// Nach der Anwahl des Referenziertyps "Fliegendes Referenzieren", 
				// ein Zyklus später kann das Referenzieren gestartet
				IF (siRefTypCyc = 0) THEN
					siRefTypCyc := siRefTypCyc + 1;
				ELSE
					// Referenzieren starten
					//sxSendBuf.sxSTW1.RefStart := True;
					sxSendBuf.STW1.x16b.bBit11 := True;
				END_IF;
			END_IF;
		END_IF;
	ELSE
		// Werte wieder zurücknehmen
	
		(*sxSendBuf.sxSTW1.Off1          := Off1;
			  sxSendBuf.sxSTW1.RejTrvTsk     := False;
			  sxSendBuf.sxSTW1.TrvStart      := False;
			  sxSendBuf.sxEPosSTW1.MdiStart  := False;
			  sxSendBuf.sxSTW1.Jog1          := False;
			  sxSendBuf.sxSTW1.Jog2          := False;
			  sxSendBuf.sxEPosSTW1.MdiTyp    := False;
			  sxSendBuf.sxEPosSTW1.MdiPos    := False;
			  sxSendBuf.sxEPosSTW1.MdiNeg    := False;
			  sxSendBuf.sxEPosSTW1.MdiTrTyp  := False;
			  sxSendBuf.sxEPosSTW1.MdiSetup  := False;
			  sxSendBuf.sxEPosSTW2.SetRefPt  := False;
			  sxSendBuf.sxEPosSTW2.RefTyp    := False;
			  sxSendBuf.sxEPosSTW2.RefStDi   := False;
			  sxSendBuf.sxEPosSTW2.JogInc    := False;
			  sxSendBuf.sxSTW1.RefStart      := False;*)
	
		sxSendBuf.STW1.x16b.bBit0		:= EnableAxis;
		sxSendBuf.STW1.x16b.bBit4		:= False;
		sxSendBuf.STW1.x16b.bBit6		:= False;
		sxSendBuf.EPosSTW1.x16b.bBit15	:= False;
		sxSendBuf.STW1.x16b.bBit8		:= False;
		sxSendBuf.STW1.x16b.bBit9		:= False;
		sxSendBuf.EPosSTW1.x16b.bBit8	:= False;
		sxSendBuf.EPosSTW1.x16b.bBit9	:= False;
		sxSendBuf.EPosSTW1.x16b.bBit10	:= False;
		sxSendBuf.EPosSTW1.x16b.bBit12	:= False;
		sxSendBuf.EPosSTW1.x16b.bBit14	:= False;
		sxSendBuf.EPosSTW2.x16b.bBit1	:= False;
		sxSendBuf.EPosSTW2.x16b.bBit8	:= False;
		sxSendBuf.EPosSTW2.x16b.bBit9	:= False;
		sxSendBuf.EPosSTW2.x16b.bBit5	:= False;
		sxSendBuf.STW1.x16b.bBit11		:= False;
	END_IF; // Hauptbetriebsart "Verfahrsätze" (Traversing Blocks)
	
	//Den Eingang ConfigEPos auf die einzelnen Bits im Telegramm verschalten
	sxSendBuf.STW1.x16b.bBit1		:= ConfigEPos.x16b.bBit0;
	sxSendBuf.STW1.x16b.bBit2		:= ConfigEPos.x16b.bBit1;
	sxSendBuf.EPosSTW2.x16b.bBit14	:= ConfigEPos.x16b.bBit2;
	sxSendBuf.EPosSTW2.x16b.bBit15	:= ConfigEPos.x16b.bBit3;
	sxSendBuf.EPosSTW2.x16b.bBit11	:= ConfigEPos.x16b.bBit4;
	sxSendBuf.EPosSTW2.x16b.bBit10	:= ConfigEPos.x16b.bBit5;
	sxSendBuf.EPosSTW2.x16b.bBit2	:= ConfigEPos.x16b.bBit6;
	sxSendBuf.STW1.x16b.bBit13		:= ConfigEPos.x16b.bBit7;
	sxSendBuf.EPosSTW1.x16b.bBit12	:= ConfigEPos.x16b.bBit8;
	sxSendBuf.STW2.x16b.bBit0		:= ConfigEPos.x16b.bBit9;
	sxSendBuf.STW2.x16b.bBit1		:= ConfigEPos.x16b.bBit10;
	sxSendBuf.STW2.x16b.bBit2		:= ConfigEPos.x16b.bBit11;
	sxSendBuf.STW2.x16b.bBit3		:= ConfigEPos.x16b.bBit12;
	sxSendBuf.STW2.x16b.bBit4		:= ConfigEPos.x16b.bBit13;
	sxSendBuf.STW2.x16b.bBit7		:= ConfigEPos.x16b.bBit14;
	sxSendBuf.STW1.x16b.bBit14		:= ConfigEPos.x16b.bBit15;
	sxSendBuf.STW1.x16b.bBit15		:= ConfigEPos2.x16b.bBit0;
	sxSendBuf.EPosSTW1.x16b.bBit6	:= ConfigEPos2.x16b.bBit1;
	sxSendBuf.EPosSTW1.x16b.bBit7	:= ConfigEPos2.x16b.bBit2;
	sxSendBuf.EPosSTW1.x16b.bBit11	:= ConfigEPos2.x16b.bBit3;
	sxSendBuf.EPosSTW1.x16b.bBit13	:= ConfigEPos2.x16b.bBit4;
	sxSendBuf.EPosSTW2.x16b.bBit3	:= ConfigEPos2.x16b.bBit5;
	sxSendBuf.EPosSTW2.x16b.bBit4	:= ConfigEPos2.x16b.bBit6;
	sxSendBuf.EPosSTW2.x16b.bBit6	:= ConfigEPos2.x16b.bBit7;
	sxSendBuf.EPosSTW2.x16b.bBit7	:= ConfigEPos2.x16b.bBit8;
	sxSendBuf.EPosSTW2.x16b.bBit12	:= ConfigEPos2.x16b.bBit9;
	sxSendBuf.EPosSTW2.x16b.bBit13	:= ConfigEPos2.x16b.bBit10;
	sxSendBuf.STW2.x16b.bBit5		:= ConfigEPos2.x16b.bBit11;
	sxSendBuf.STW2.x16b.bBit6		:= ConfigEPos2.x16b.bBit12;
	sxSendBuf.STW2.x16b.bBit8		:= ConfigEPos2.x16b.bBit13;
	sxSendBuf.STW2.x16b.bBit9		:= ConfigEPos2.x16b.bBit14;
	
	swSendBuf[0]	:= sxSendBuf.STW1.ui16b;
	swSendBuf[1]	:= sxSendBuf.EPosSTW1.ui16b;
	swSendBuf[2]	:= sxSendBuf.EPosSTW2.ui16b;
	swSendBuf[3]	:= sxSendBuf.STW2.ui16b;
	swSendBuf[4]	:= sxSendBuf.OverrideV;
	swSendBuf[5]	:= sxSendBuf.Position.uints[1];	//    %W1;
	swSendBuf[6]	:= sxSendBuf.Position.uints[0];	//	%W0;
	swSendBuf[7]	:= sxSendBuf.Velocity.uints[1];	// 
	swSendBuf[8]	:= sxSendBuf.Velocity.uints[0];	//
	swSendBuf[9]	:= sxSendBuf.OverrideA;
	swSendBuf[10]	:= sxSendBuf.OverrideD;
	swSendBuf[11]	:= sxSendBuf.Reserve;
	
	//Prozessdaten zur Signalbaugruppe schreiben
	piRetSFC := 0;
	//DPWR_DAT(LADDR := HWIDSTW,RECORD := swSendBuf);
	
	HWIDSTW.StatusWord0.ui16b	:= swSendBuf[0];
	HWIDSTW.StatusWord1.ui16b	:= swSendBuf[1];
	HWIDSTW.StatusWord2.ui16b	:= swSendBuf[2];
	HWIDSTW.StatusWord3.ui16b	:= swSendBuf[3];
	HWIDSTW.StatusWord4.ui16b	:= swSendBuf[4];
	HWIDSTW.StatusWord5.ui16b	:= swSendBuf[5];
	HWIDSTW.StatusWord6.ui16b	:= swSendBuf[6];
	HWIDSTW.StatusWord7.ui16b	:= swSendBuf[7];
	HWIDSTW.StatusWord8.ui16b	:= swSendBuf[8];
	HWIDSTW.StatusWord9.ui16b	:= swSendBuf[9];
	HWIDSTW.StatusWord10.ui16b	:= swSendBuf[10];
	HWIDSTW.StatusWord11.ui16b	:= swSendBuf[11];
	
	// Fehler der Rückmeldung ausgeben
	DiagID := INT_TO_WORD(piRetSFC);
	
	//kein Fehler beim Schreiben
	IF piRetSFC = 0 THEN
	
		// Fehler wieder zurück nehmen
		IF (swStatus = 16#8601) THEN
			swStatus	:= 16#7002;
			Error		:= False;
		END_IF;
	
		//Prozessdaten von der Signalbaugruppe lesen
		piRetSFC := 0;
		//DPRD_DAT(LADDR := HWIDZSW,RECORD => swRecvBuf);
	
		swRecvBuf[0]	:= HWIDZSW.StatusWord0.ui16b;
		swRecvBuf[1]	:= HWIDZSW.StatusWord1.ui16b;
		swRecvBuf[2]	:= HWIDZSW.StatusWord2.ui16b;
		swRecvBuf[3]	:= HWIDZSW.StatusWord3.ui16b;
		swRecvBuf[4]	:= HWIDZSW.StatusWord4.ui16b;
		swRecvBuf[5]	:= HWIDZSW.StatusWord5.ui16b;
		swRecvBuf[6]	:= HWIDZSW.StatusWord6.ui16b;
		swRecvBuf[7]	:= HWIDZSW.StatusWord7.ui16b;
		swRecvBuf[8]	:= HWIDZSW.StatusWord8.ui16b;
		swRecvBuf[9]	:= HWIDZSW.StatusWord9.ui16b;
		swRecvBuf[10]	:= HWIDZSW.StatusWord10.ui16b;
		swRecvBuf[11]	:= HWIDZSW.StatusWord11.ui16b;
	
		// Fehlermeldung der Rückmeldung ausgeben
		DiagID := INT_TO_WORD(piRetSFC);
	
		//Fehler beim Lesen (Profibus-Kommunikation unterbrochen)
		IF piRetSFC <> 0 THEN
	
			// Fehler
			Error		:= TRUE;
			swStatus	:= 16#8600;
	
			// Zustandsworte löschen
			sxRecvBuf.ZSW1.ui16b		:= 0;
			sxRecvBuf.EPosZSW1.ui16b	:= 0;
			sxRecvBuf.EPosZSW2.ui16b	:= 0;
			sxRecvBuf.ZSW2.ui16b		:= 0;
			sxRecvBuf.NotUsed			:= 0;
			sxRecvBuf.Position.Valor	:= 0;
			sxRecvBuf.Velocity.Valor	:= 0;
			sxRecvBuf.ErrNr				:= 0;
			sxRecvBuf.WarnNr			:= 0;
			sxRecvBuf.Reserve			:= 0;
	
			// Werte auslesen
		ELSE
	
			// Fehler wieder zurück nehmen
			IF (swStatus = 16#8600) THEN
				swStatus	:= 16#7002;
				Error		:= False;
			END_IF;
	
			sxRecvBuf.ZSW1.ui16b		:= swRecvBuf[0];
			sxRecvBuf.EPosZSW1.ui16b	:= swRecvBuf[1];
			sxRecvBuf.EPosZSW2.ui16b	:= swRecvBuf[2];
			sxRecvBuf.ZSW2.ui16b		:= swRecvBuf[3];
			sxRecvBuf.NotUsed			:= swRecvBuf[4];
			sxRecvBuf.Position.uints[1]	:= swRecvBuf[5];
			sxRecvBuf.Position.uints[0]	:= swRecvBuf[6];
			sxRecvBuf.Velocity.uints[1]	:= swRecvBuf[7];
			sxRecvBuf.Velocity.uints[0]	:= swRecvBuf[8];
			sxRecvBuf.ErrNr				:= swRecvBuf[9];
			sxRecvBuf.WarnNr			:= swRecvBuf[10];
			sxRecvBuf.Reserve			:= swRecvBuf[11];
	
			// ZSW1 aufbereiten
			//Busy := sxRecvBuf.sxZSW1.IOp;
			sbBusy := sxRecvBuf.ZSW1.x16b.bBit2;
	
			// Fehler auswerten
	
			(*IF sxRecvBuf.sxZSW1.Fault THEN
					  ErrorId := 5;
					  Error := True;
				  ELSIF sxRecvBuf.sxZSW1.PowInhbt THEN 
					  ErrorId := 6;
					  Error := True;
				  ELSE
					  // Fehler wieder zurück nehmen
					  IF (ErrorId = 5) OR (ErrorId = 6) THEN
						  ErrorId := 0;    
						  Error := False;
					  END_IF;
				  END_IF;*)
	
			IF sxRecvBuf.ZSW1.x16b.bBit3 THEN
				swStatus	:= 16#8401;
				Error		:= True;
			ELSIF sxRecvBuf.ZSW1.x16b.bBit6 THEN
				swStatus	:= 16#8402;
				Error		:= True;
			ELSE
				// Fehler wieder zurück nehmen
				IF (swStatus = 16#8401) OR (swStatus = 16#8402) THEN
					swStatus	:= 16#7002;
					Error		:= False;
				END_IF;
			END_IF;
	
			// EPOS_ZSW1            
			// EPOS-Wort-1 BIT 00 --> 1 = Active traversing block bit 0
			//IF sxRecvBuf.sxEPosZSW1.ActTrvBit0 THEN
			IF sxRecvBuf.EPosZSW1.x16b.bBit0 THEN
				swEPosZSW1 := swEPosZSW1 OR 16#01;
			ELSE
				swEPosZSW1 := swEPosZSW1 AND 16#FFFE;
			END_IF;
	
			// EPOS-Wort-1 Bit 01 --> 1 = Active traversing block bit 1
			//IF sxRecvBuf.sxEPosZSW1.ActTrvBit1 THEN
			IF sxRecvBuf.EPosZSW1.x16b.bBit1 THEN
				swEPosZSW1 := swEPosZSW1 OR 16#02;
			ELSE
				swEPosZSW1 := swEPosZSW1 AND 16#FFFD;
			END_IF;
	
			// EPOS-Wort-1 Bit 02 --> 1 = Active traversing block bit 2
			//IF sxRecvBuf.sxEPosZSW1.ActTrvBit2 THEN
			IF sxRecvBuf.EPosZSW1.x16b.bBit2 THEN
				swEPosZSW1 := swEPosZSW1 OR 16#04;
			ELSE
				swEPosZSW1 := swEPosZSW1 AND 16#FFFB;
			END_IF;
	
			// EPOS-Wort-1 Bit 03 --> 1 = Active traversing block bit 3
			//IF sxRecvBuf.sxEPosZSW1.ActTrvBit3 THEN
			IF sxRecvBuf.EPosZSW1.x16b.bBit3 THEN
				swEPosZSW1 := swEPosZSW1 OR 16#08;
			ELSE
				swEPosZSW1 := swEPosZSW1 AND 16#FFF7;
			END_IF;
	
			// EPOS-Wort-1 Bit 04 --> 1 = Active traversing block bit 4 
			//IF sxRecvBuf.sxEPosZSW1.ActTrvBit4 THEN
			IF sxRecvBuf.EPosZSW1.x16b.bBit4 THEN
				swEPosZSW1 := swEPosZSW1 OR 16#10;
			ELSE
				swEPosZSW1 := swEPosZSW1 AND 16#FFEF;
			END_IF;
	
			// EPOS-Wort-1 Bit 05 --> 1 = Active traversing block bit 5
			//IF sxRecvBuf.sxEPosZSW1.ActTrvBit5 THEN
			IF sxRecvBuf.EPosZSW1.x16b.bBit5 THEN
				swEPosZSW1 := swEPosZSW1 OR 16#20;
			ELSE
				swEPosZSW1 := swEPosZSW1 AND 16#FFDF;
			END_IF;
	
			// EPOS-Wort-1 Bit 08 --> 1 = STOP cam minus active
			//IF sxRecvBuf.sxEPosZSW1.StpCamMinAct THEN
			IF sxRecvBuf.EPosZSW1.x16b.bBit8 THEN
				swEPosZSW1 := swEPosZSW1 OR 16#100;
			ELSE
				swEPosZSW1 := swEPosZSW1 AND 16#FEFF;
			END_IF;
	
			// EPOS-Wort-1 Bit 09 --> 1 = STOP cam plus active
			//IF sxRecvBuf.sxEPosZSW1.StpCamPlsAct THEN
			IF sxRecvBuf.EPosZSW1.x16b.bBit9 THEN
				swEPosZSW1 := swEPosZSW1 OR 16#200;
			ELSE
				swEPosZSW1 := swEPosZSW1 AND 16#FDFF;
			END_IF;
	
			// EPOS-Wort-1 Bit 10 --> 1 = Jogging active
			//IF sxRecvBuf.sxEPosZSW1.JogAct THEN
			IF sxRecvBuf.EPosZSW1.x16b.bBit10 THEN
				swEPosZSW1 := swEPosZSW1 OR 16#400;
			ELSE
				swEPosZSW1 := swEPosZSW1 AND 16#FBFF;
			END_IF;
	
			// EPOS-Wort-1 Bit 11 --> 1 = Reference point approach active
			//IF sxRecvBuf.sxEPosZSW1.RefAct THEN
			IF sxRecvBuf.EPosZSW1.x16b.bBit11 THEN
				swEPosZSW1 := swEPosZSW1 OR 16#800;
			ELSE
				swEPosZSW1 := swEPosZSW1 AND 16#F7FF;
			END_IF;
	
			// Anstossen des fliegenden Referenzieren prüfen, wenn die Rückmeldung fehlt dann wiederholen
			//IF NOT sxRecvBuf.sxEPosZSW1.FlyRefAct AND sbRefTyp AND sxSendBuf.sxSTW1.RefStart THEN
			IF NOT sxRecvBuf.EPosZSW1.x16b.bBit12 AND sbRefTyp AND sxSendBuf.STW1.x16b.bBit11 THEN
	
				// Wiederholung anstossen 
				IF siRefActRetry < siRetryMax THEN
					siRefActRetry := siRefActRetry + 1;
	
					// Referenzieren starten wieder wegnehmen
					//sxSendBuf.sxSTW1.RefStart := False;
					sxSendBuf.STW1.x16b.bBit11 := False;
				ELSE
	
					// Fehlermeldung
					swStatus	:= 16#8403;
					Error		:= True;
				END_IF;
			ELSE
	
				// Fehler wieder zurücknehmen, wenn er mal ausgelöst wurde
				IF swStatus = 16#8403 THEN
					swStatus	:= 16#7002;
					Error		:= False;
				END_IF;
			END_IF;
	
			// EPOS-Wort-1 Bit 12 --> 1 = Flying referencing active
			//IF sxRecvBuf.sxEPosZSW1.FlyRefAct THEN
			IF sxRecvBuf.EPosZSW1.x16b.bBit12 THEN
				swEPosZSW1 := swEPosZSW1 OR 16#1000;
			ELSE
				swEPosZSW1 := swEPosZSW1 AND 16#EFFF;
			END_IF;
	
			// EPOS-Wort-1 Bit 13 --> 1 = Traversing block active
			//IF sxRecvBuf.sxEPosZSW1.TrvBlAct THEN
			IF sxRecvBuf.EPosZSW1.x16b.bBit13 THEN
				swEPosZSW1 := swEPosZSW1 OR 16#2000;
			ELSE
				swEPosZSW1 := swEPosZSW1 AND 16#DFFF;
			END_IF;
	
			// EPOS-Wort-1 Bit 14 --> 1 = MDI setup active
			//IF sxRecvBuf.sxEPosZSW1.MdiStupAct THEN
			IF sxRecvBuf.EPosZSW1.x16b.bBit14 THEN
				swEPosZSW1 := swEPosZSW1 OR 16#4000;
			ELSE
				swEPosZSW1 := swEPosZSW1 AND 16#BFFF;
			END_IF;
	
			// EPOS-Wort-1 Bit 15 --> 1 = MDI positing active
			//IF sxRecvBuf.sxEPosZSW1.MdiPosAct THEN
			IF sxRecvBuf.EPosZSW1.x16b.bBit15 THEN
				swEPosZSW1 := swEPosZSW1 OR 16#8000;
			ELSE
				swEPosZSW1 := swEPosZSW1 AND 16#7FFF;
			END_IF;
	
			// EPOS_ZSW2 
			// EPOS-Wort-2 Bit 00 --> 1 = Tracking mode active
			//IF sxRecvBuf.sxEPosZSW2.TrkModeAct THEN
			IF sxRecvBuf.EPosZSW2.x16b.bBit0 THEN
				swEPosZSW2 := swEPosZSW2 OR 16#01;
			ELSE
				swEPosZSW2 := swEPosZSW2 AND 16#FFFE;
			END_IF;
	
			// EPOS-Wort-2 Bit 01 --> 1 = Velocity limit active
			//IF sxRecvBuf.sxEPosZSW2.VeloLimAct THEN
			IF sxRecvBuf.EPosZSW2.x16b.bBit1 THEN
				swEPosZSW2 := swEPosZSW2 OR 16#02;
			ELSE
				swEPosZSW2 := swEPosZSW2 AND 16#FFFD;
			END_IF;
	
			// EPOS-Wort-2 Bit 02 --> 1 = Setpoint static
			//IF sxRecvBuf.sxEPosZSW2.SetPStat THEN
			IF sxRecvBuf.EPosZSW2.x16b.bBit2 THEN
				swEPosZSW2 := swEPosZSW2 OR 16#04;
			ELSE
				swEPosZSW2 := swEPosZSW2 AND 16#FFFB;
			END_IF;
	
			// EPOS-Wort-2 Bit 03 --> 1 = Printmark outside outer window
			//IF sxRecvBuf.sxEPosZSW2.PrnMrkOut THEN
			IF sxRecvBuf.EPosZSW2.x16b.bBit3 THEN
				swEPosZSW2 := swEPosZSW2 OR 16#08;
			ELSE
				swEPosZSW2 := swEPosZSW2 AND 16#FFF7;
			END_IF;
	
			// EPOS-Wort-2 Bit 04 --> 1 = Axis forwards
			//IF sxRecvBuf.sxEPosZSW2.FWD THEN
			IF sxRecvBuf.EPosZSW2.x16b.bBit4 THEN
				swEPosZSW2 := swEPosZSW2 OR 16#10;
			ELSE
				swEPosZSW2 := swEPosZSW2 AND 16#FFEF;
			END_IF;
	
			// EPOS-Wort-2 Bit 05 --> 1 = Axis backwards
			//IF sxRecvBuf.sxEPosZSW2.BWD THEN
			IF sxRecvBuf.EPosZSW2.x16b.bBit5 THEN
				swEPosZSW2 := swEPosZSW2 OR 16#20;
			ELSE
				swEPosZSW2 := swEPosZSW2 AND 16#FFDF;
			END_IF;
	
			// EPOS-Wort-2 Bit 06 --> 1 = Software limit switch minus active
			//IF sxRecvBuf.sxEPosZSW2.SftSwMinAct THEN
			IF sxRecvBuf.EPosZSW2.x16b.bBit6 THEN
				swEPosZSW2 := swEPosZSW2 OR 16#40;
			ELSE
				swEPosZSW2 := swEPosZSW2 AND 16#FFBF;
			END_IF;
	
			// EPOS-Wort-2 Bit 07 --> 1 = Software limit switch plus active
			//IF sxRecvBuf.sxEPosZSW2.SftSwPlsAct THEN
			IF sxRecvBuf.EPosZSW2.x16b.bBit7 THEN
				swEPosZSW2 := swEPosZSW2 OR 16#80;
			ELSE
				swEPosZSW2 := swEPosZSW2 AND 16#FF7F;
			END_IF;
	
			// EPOS-Wort-2 Bit 08 --> 1 = Position actual value <= cam position 1
			//IF sxRecvBuf.sxEPosZSW2.PosSmCam1 THEN
			IF sxRecvBuf.EPosZSW2.x16b.bBit8 THEN
				swEPosZSW2 := swEPosZSW2 OR 16#100;
			ELSE
				swEPosZSW2 := swEPosZSW2 AND 16#FEFF;
			END_IF;
	
			// EPOS-Wort-2 Bit 09 --> 1 = Position actual value <= cam position 2
			//IF sxRecvBuf.sxEPosZSW2.PosSmCam2 THEN
			IF sxRecvBuf.EPosZSW2.x16b.bBit9 THEN
				swEPosZSW2 := swEPosZSW2 OR 16#200;
			ELSE
				swEPosZSW2 := swEPosZSW2 AND 16#FDFF;
			END_IF;
	
			// EPOS-Wort-2 Bit 10 --> 1 = Direct output 1 via traversing block
			//IF sxRecvBuf.sxEPosZSW2.TrvOut1 THEN
			IF sxRecvBuf.EPosZSW2.x16b.bBit10 THEN
				swEPosZSW2 := swEPosZSW2 OR 16#400;
			ELSE
				swEPosZSW2 := swEPosZSW2 AND 16#FBFF;
			END_IF;
	
			// EPOS-Wort-2 Bit 11 --> 1 = Direct output 2 via traversing block
			//IF sxRecvBuf.sxEPosZSW2.TrvOut2 THEN
			IF sxRecvBuf.EPosZSW2.x16b.bBit11 THEN
				swEPosZSW2 := swEPosZSW2 OR 16#800;
			ELSE
				swEPosZSW2 := swEPosZSW2 AND 16#F7FF;
			END_IF;
	
			// EPOS-Wort-2 Bit 12 --> 1 = Fixed STOP reached
			//IF sxRecvBuf.sxEPosZSW2.FxStpRd THEN
			IF sxRecvBuf.EPosZSW2.x16b.bBit12 THEN
				swEPosZSW2 := swEPosZSW2 OR 16#1000;
			ELSE
				swEPosZSW2 := swEPosZSW2 AND 16#EFFF;
			END_IF;
	
			// EPOS-Wort-2 Bit 13 --> 1 = Fixed STOP clamping torque reached
			//IF sxRecvBuf.sxEPosZSW2.FxStpTrRd THEN
			IF sxRecvBuf.EPosZSW2.x16b.bBit13 THEN
				swEPosZSW2 := swEPosZSW2 OR 16#2000;
			ELSE
				swEPosZSW2 := swEPosZSW2 AND 16#DFFF;
			END_IF;
	
			// EPOS-Wort-2 Bit 14 --> 1 = Traversing fixed STOP active
			//IF sxRecvBuf.sxEPosZSW2.TrvFxStpAct THEN
			IF sxRecvBuf.EPosZSW2.x16b.bBit14 THEN
				swEPosZSW2 := swEPosZSW2 OR 16#4000;
			ELSE
				swEPosZSW2 := swEPosZSW2 AND 16#BFFF;
			END_IF;
	
			// EPOS-Wort-2 Bit 15 --> 1 = Traversing command active
			//IF sxRecvBuf.sxEPosZSW2.CmdAct THEN
			IF sxRecvBuf.EPosZSW2.x16b.bBit15 THEN
				swEPosZSW2 := swEPosZSW2 OR 16#8000;
			ELSE
				swEPosZSW2 := swEPosZSW2 AND 16#7FFF;
			END_IF;
	
			sbReady := sxRecvBuf.ZSW1.x16b.bBit1;
	
			AxisEnabled	:= sxRecvBuf.ZSW1.x16b.bBit2;
			sbIOp		:= sxRecvBuf.ZSW1.x16b.bBit2;
	
			AxisError	:= sxRecvBuf.ZSW1.x16b.bBit3;
			sbFault		:= sxRecvBuf.ZSW1.x16b.bBit3;
	
			AxisWarn	:= sxRecvBuf.ZSW1.x16b.bBit7;
			sbAlarm		:= sxRecvBuf.ZSW1.x16b.bBit7;
	
			AxisPosOk	:= sxRecvBuf.ZSW1.x16b.bBit10;
			AxisRef		:= sxRecvBuf.ZSW1.x16b.bBit11;
	
			sbAccel	:= sxRecvBuf.ZSW1.x16b.bBit14;
			sbDecel	:= sxRecvBuf.ZSW1.x16b.bBit15;
	
			ActVelocity	:= DWORD_TO_DINT(sxRecvBuf.Velocity.Valor);
			ActPosition	:= DWORD_TO_DINT(sxRecvBuf.Position.Valor);
			ActMode		:= ModePos;
			ActWarn		:= sxRecvBuf.WarnNr;
			ActFault	:= sxRecvBuf.ErrNr;
	
			Lockout := sxRecvBuf.ZSW1.x16b.bBit6;
		END_IF;
	ELSE
	
		// Fehler
		Error		:= TRUE;
		swStatus	:= 16#8601;
	
	END_IF;
	
	// Initialisierung von Ausg㭧en
	Status		:= swStatus;
	EPosZSW1	:= swEPosZSW1;
	EPosZSW2	:= swEPosZSW2;
	
ELSE
	ValidaLicensa();
END_IF

END_FUNCTION_BLOCK

// POUs/PRG_TEST
PROGRAM PRG_TEST
VAR CONSTANT
	aux : INT := 50;
END_VAR

VAR
	

	fb1 : fb_Partida;
	fb2 : FB_ComunicacaoCanOpen;
	fb3 : FB_ComunicacaoEthernet;
	fb4 : FB_DeltaMS;
	fb5 : FB_ModBusRTU_AC380;
	fb6 : FB_ModBusRTU_ALTISTAR22;
	fb7 : FB_ModBusRTU_ATV320;
	fb8 : Sina_posV2;
	fb9 : Sina_SpeedV2;
	fb10 : ARRAY[1..2] OF FB_Comunicacao_AX5000;
	fb11 : FB_TeSysU_Can;
	
	ReferenciaAxis : ARRAY[1..2] OF AXIS_REF;




	FBPartida_Test : fb_partida_teste;

	linkObrigatorio AT %I* : UINT;

	stAux : st_SinaSpeed;
	//FBmotor : Sina_SpeedV2;
	i	: INT;
	j	: INT;

	stAux1		: ARRAY[1..10] OF st_SinaSpeed;
	FBmotor1	: ARRAY[1..10] OF Sina_SpeedV2;

	partidaSimples : FB_Partida;

	partida		: ARRAY[0..10] OF FB_Partida;
	EthernetCOM	: FB_ComunicacaoEthernet;

	partidas	: ARRAY[1..aux] OF FB_Partida;
	stPartidas	: ARRAY[1..aux] OF st_Partida;

	rLSP				: REAL;	//velocidade minima
	rHSP				: REAL;	//velocidade maxima
	rTRF				: REAL;	//maxima velocidade
	rITH				: REAL;	//corrente maxima 
	rACC				: REAL;	//rampa de aceleração
	rDEC				: REAL;	//rampa de desaceleração
	xPHR				: BOOL;	//ordem das fases
	xEscreveParametros	: BOOL;
	xLerParametros		: BOOL;

	CAN : ARRAY[0..10] OF FB_ComunicacaoCanOpen;

	ITH_E	: REAL;	//corrente maxima 
	ACC_E	: REAL;	//rampa de aceleração
	DEC_E	: REAL;	//rampa de desaceleração
	PHR_E	: BOOL;	//ordem das fases

	xEscreve1	: BOOL;
	xEscreve2	: BOOL;
	xEscreve3	: BOOL;


	fbGeral : FB_SalvaPersistentesEHoraAgora;

	configCAN : ARRAY[1..5] OF Config_CAN;

	LinkCan : ARRAY[1..5] OF ATV320_Can;

	xLe : BOOL;

	fbWritePersistent	: FB_WritePersistentData;
	xStart				: BOOL;

	xTeste1	: LREAL;
	xTeste2	: BOOL;
	
	MestreCan1 AT %I* : AMSNETID;

	xParteTodos : BOOL;
	
	partidaDelta : st_Partida;
	fbPartida : FB_Partida;
	fbDelta : FB_DeltaMS;
	linkDelta : st_LinkDeltaEIP;
	
	emergenciaAux : BOOL := TRUE;
	
	rtLigou : R_TRIG;
	rtChegou : R_TRIG;
	tempoAgora : TIME;
	tempoqueDemorou : TIME;
	tAux : TIME;
	
	rtLigou2 : R_TRIG;
	rtChegou2 : R_TRIG;
	tempoAgora2 : TIME;
	tempoqueDemorou2 : TIME;
	
	
	
	stPartida	: ARRAY[0..200] OF st_Partida;
	fbPartida2	: ARRAY[0..200] OF fb_partida;
	stPartida2	: ARRAY[0..200] OF st_Partida;
	
	
	PartidasRodando : INT;
	
	fbSinaSpeed : Sina_SpeedV2;
	
	xForca3s : BOOL;

END_VAR

VAR RETAIN PERSISTENT
	config : ConfigComunicacaoEthernet;
END_VAR

//TcUnit.RUN();
//TcUnit.RUN_IN_SEQUENCE();

fbGeral(hrAgora =>);


TesteCanTeSysU();







//TesteProfinet();
(*
IF xForca3s THEN
	stPartida[1].en.xLigaManu3S := TRUE;
END_IF
TestePartidaSimples();

*)



i := j;

ACTION Teste:
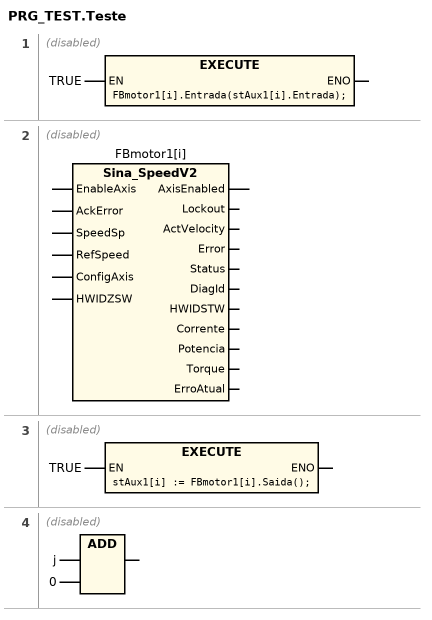
// NETWORK 1 (disabled)
// FBmotor1[i].Entrada(stAux1[i].Entrada);

// NETWORK 2 (disabled)
// FBmotor1[i](); // Sina_SpeedV2

// NETWORK 3 (disabled)
// stAux1[i] := FBmotor1[i].Saida();

// NETWORK 4 (disabled)
// (* j + 0; result not used *)
END_ACTION

ACTION TesteAX5000:
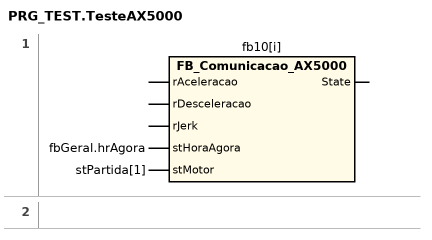
// NETWORK 1
fb10[i](stHoraAgora := fbGeral.hrAgora, stMotor := stPartida[1]); // FB_Comunicacao_AX5000

// NETWORK 2
END_ACTION

ACTION TesteCan:
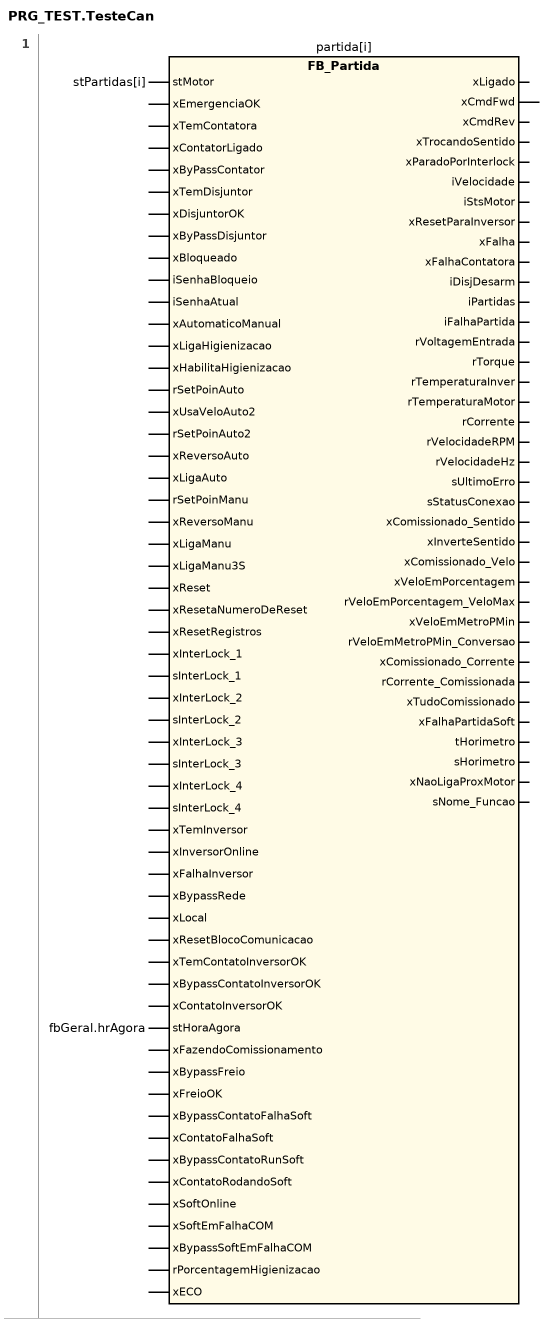
// NETWORK 1
partida[i](stMotor := stPartidas[i], stHoraAgora := fbGeral.hrAgora); // FB_Partida

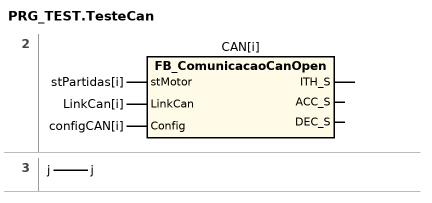
// NETWORK 2
CAN[i](stMotor := stPartidas[i], LinkCan := LinkCan[i], Config := configCAN[i]); // FB_ComunicacaoCanOpen

// NETWORK 3
j := j;
END_ACTION

ACTION TesteCanTeSysU:
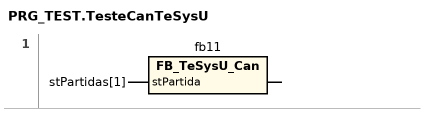
// NETWORK 1
fb11(stPartida := stPartidas[1]); // FB_TeSysU_Can

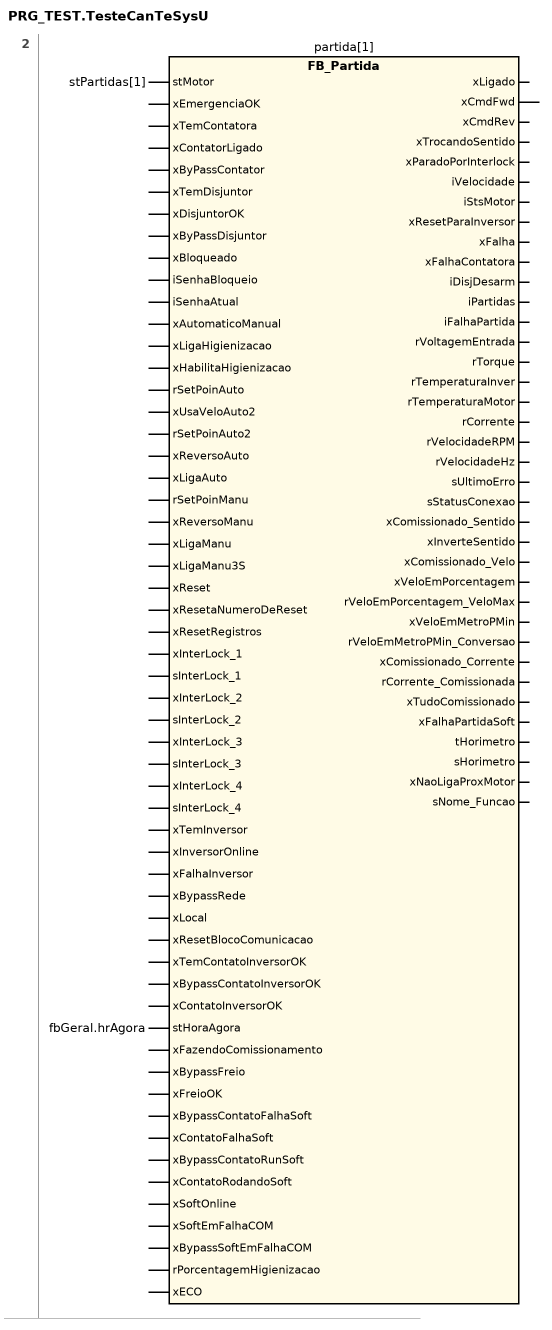
// NETWORK 2
partida[1](stMotor := stPartidas[1], stHoraAgora := fbGeral.hrAgora); // FB_Partida
END_ACTION

ACTION TesteDelta:
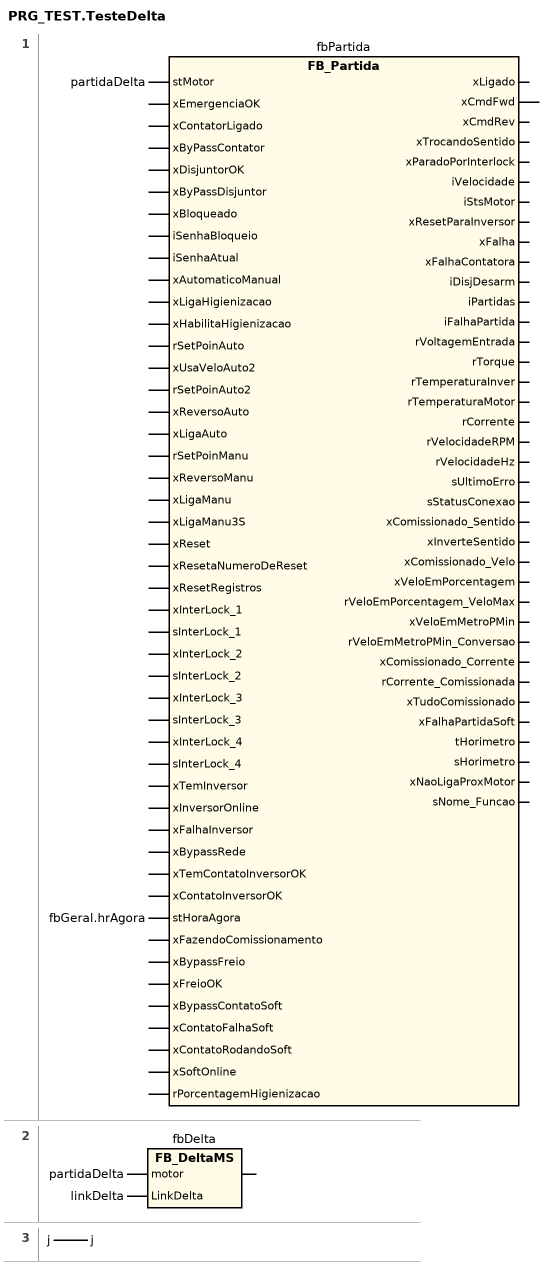
// NETWORK 1
fbPartida(stMotor := partidaDelta, stHoraAgora := fbGeral.hrAgora); // FB_Partida

// NETWORK 2
fbDelta(motor := partidaDelta, LinkDelta := linkDelta); // FB_DeltaMS

// NETWORK 3
j := j;
END_ACTION

ACTION TestePartida:
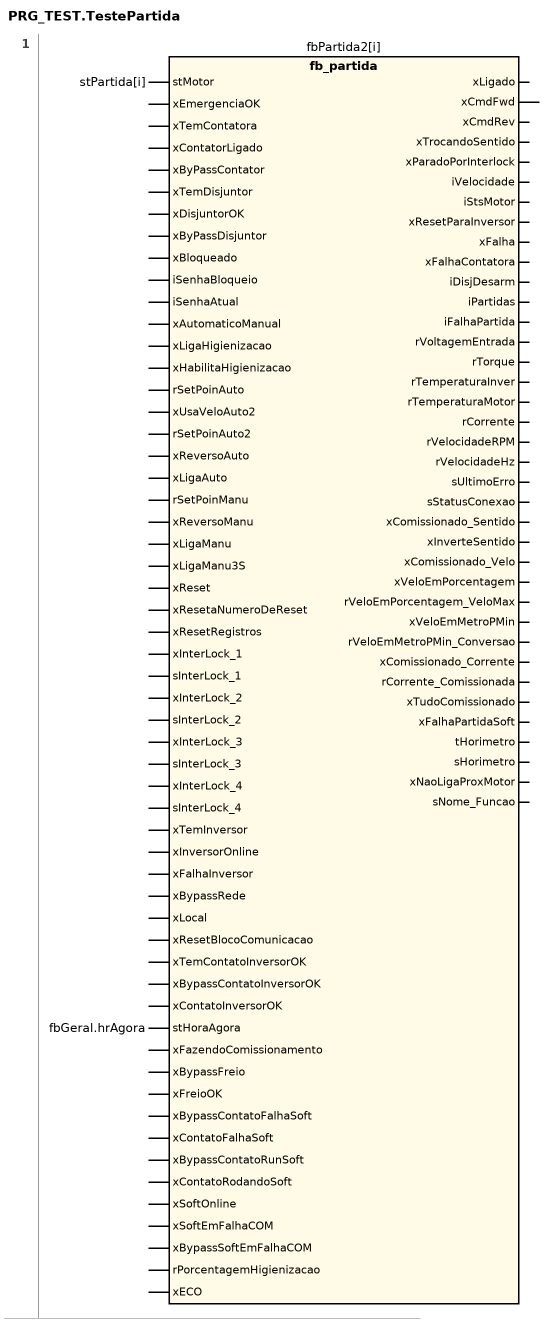
// NETWORK 1
fbPartida2[i](stMotor := stPartida[i], stHoraAgora := fbGeral.hrAgora); // fb_partida

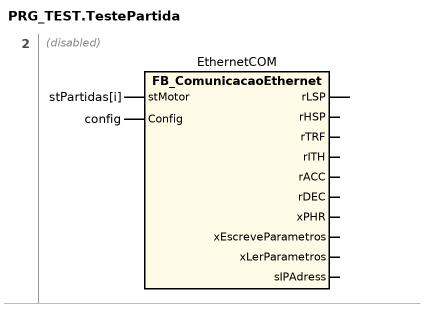
// NETWORK 2 (disabled)
// EthernetCOM(stMotor := stPartidas[i], Config := config); // FB_ComunicacaoEthernet
END_ACTION

ACTION TestePartidaSimples:
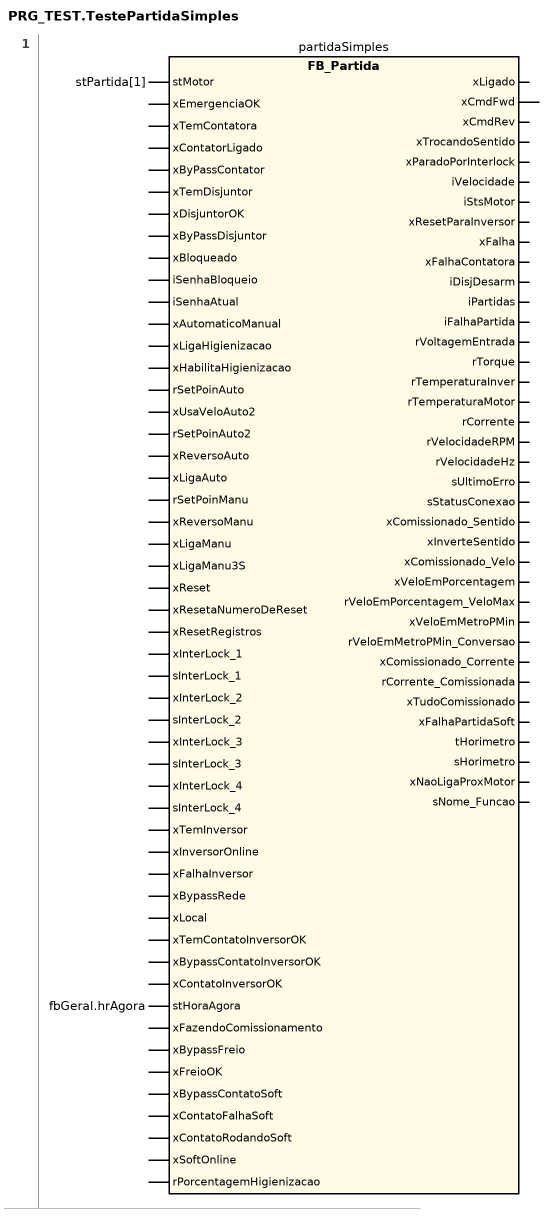
// NETWORK 1
partidaSimples(stMotor := stPartida[1], stHoraAgora := fbGeral.hrAgora); // FB_Partida
END_ACTION

ACTION TesteProfinet:
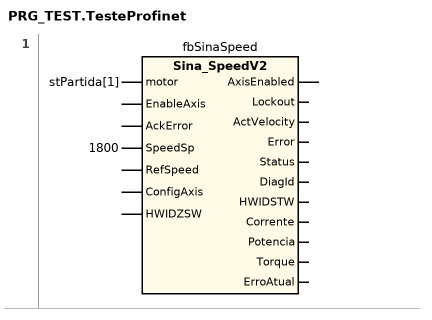
// NETWORK 1
fbSinaSpeed(motor := stPartida[1], SpeedSp := 1800); // Sina_SpeedV2

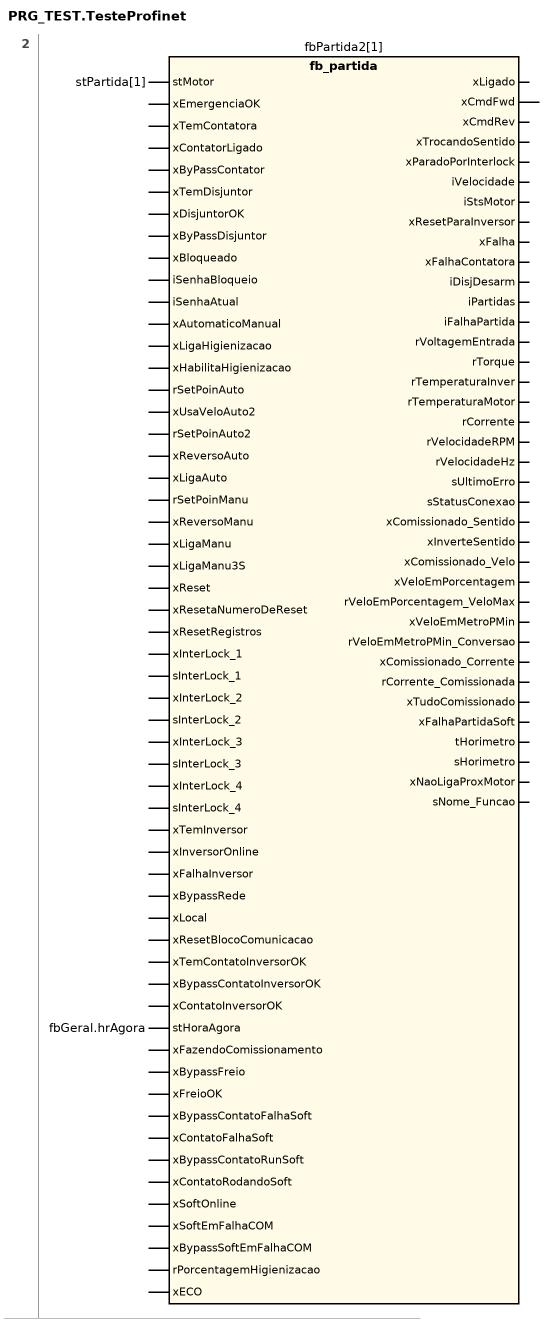
// NETWORK 2
fbPartida2[1](stMotor := stPartida[1], stHoraAgora := fbGeral.hrAgora); // fb_partida
END_ACTION

END_PROGRAM

// Project Information/F_GetCompany
// This function has been automatically generated from the project information.
{attribute 'signature_flag' := '1073741824'}
{attribute 'TcGenerated'}
{attribute 'no-analysis'}
FUNCTION F_GetCompany : WSTRING
VAR_INPUT
	
END_VAR

F_GetCompany := "Teknike";

END_FUNCTION

// Project Information/F_GetTitle
// This function has been automatically generated from the project information.
{attribute 'signature_flag' := '1073741824'}
{attribute 'TcGenerated'}
{attribute 'no-analysis'}
FUNCTION F_GetTitle : WSTRING
VAR_INPUT
	
END_VAR

F_GetTitle := "Partidas";

END_FUNCTION

// Project Information/F_GetVersion
// This function has been automatically generated from the project information.
{attribute 'signature_flag' := '1073741824'}
{attribute 'TcGenerated'}
{attribute 'no-analysis'}
FUNCTION F_GetVersion : ST_LibVersion
VAR_INPUT
	
END_VAR

F_GetVersion.iMajor := 1;
F_GetVersion.iMinor := 9;
F_GetVersion.iBuild := 11;
F_GetVersion.iRevision := 0;
F_GetVersion.sVersion := '1.9.11';
F_GetVersion.nFlags := 0;

END_FUNCTION
